DATA_BLOCK "HF4_Sum_SCtrl"	// DB 6040
VERSION : 0.1
  STRUCT
   SDPH_1_SCtrl : WORD ;
   SDPH_2_SCtrl : WORD ;
   SDPH_3_SCtrl : WORD ;
   SDPH_4_SCtrl : WORD ;
   SDPH_5_SCtrl : WORD ;
   SDPH_6_SCtrl : WORD ;
   SDPH_7_SCtrl : WORD ;
   SDPH_8_SCtrl : WORD ;
   SDPH_9_SCtrl : WORD ;
   SDPH_10_SCtrl : WORD ;
   SB_1_SCtrl : WORD ;
   SB_2_SCtrl : WORD ;
   SB_3_SCtrl : WORD ;
   SB_4_SCtrl : WORD ;
   SB_5_SCtrl : WORD ;
   SB_6_SCtrl : WORD ;
   SB_7_SCtrl : WORD ;
   SB_8_SCtrl : WORD ;
   SB_9_SCtrl : WORD ;
   SB_10_SCtrl : WORD ;
   SB_11_SCtrl : WORD ;
   SB_12_SCtrl : WORD ;
   SB_13_SCtrl : WORD ;
   SB_14_SCtrl : WORD ;
   SB_15_SCtrl : WORD ;
   SB_16_SCtrl : WORD ;
   SB_17_SCtrl : WORD ;
   SB_18_SCtrl : WORD ;
   KT_A1_SCtrl : WORD ;
   HPF_A1_SCtrl : WORD ;
   DTS_A1_SCtrl : WORD ;
   DTS_A2_SCtrl : WORD ;
   DTS_A3_SCtrl : WORD ;
   DTS_A4_SCtrl : WORD ;
   DTS_A5_SCtrl : WORD ;
   DTS_A6_SCtrl : WORD ;
   DTS_A7_SCtrl : WORD ;
   DTS_A8_SCtrl : WORD ;
   DTS_A9_SCtrl : WORD ;
   DTS_A10_SCtrl : WORD ;
   TVF_A1_SCtrl : WORD ;
   TVF_A2_SCtrl : WORD ;
   UOF_A1_SCtrl : WORD ;
   DM_A1_SCtrl : WORD ;
   DM_A2_SCtrl : WORD ;
   DM_A3_SCtrl : WORD ;
   DM_A4_SCtrl : WORD ;
   DM_A5_SCtrl : WORD ;
   DM_A6_SCtrl : WORD ;
   DM_A7_SCtrl : WORD ;
   DM_A8_SCtrl : WORD ;
   DM_A9_SCtrl : WORD ;
   DM_A10_SCtrl : WORD ;
   U0F_DT_A1_SCtrl : WORD ;
   U0F_DT_A2_SCtrl : WORD ;
   U0F_DT_A3_SCtrl : WORD ;
   U0F_DT_A4_SCtrl : WORD ;
   U0F_DT_A5_SCtrl : WORD ;
   U0F_DT_A6_SCtrl : WORD ;
   K1_XK_A1_SCtrl : WORD ;
   K1_HPF_A1_SCtrl : WORD ;
   K1_DTS_A1_SCtrl : WORD ;
   K1_DTS_A2_SCtrl : WORD ;
   K1_DTS_A3_SCtrl : WORD ;
   K2_XK_A1_SCtrl : WORD ;
   K2_HPF_A1_SCtrl : WORD ;
   K2_DTS_A1_SCtrl : WORD ;
   K2_DTS_A2_SCtrl : WORD ;
   K2_DTS_A3_SCtrl : WORD ;
   K3_XK_A1_SCtrl : WORD ;
   K3_HPF_A1_SCtrl : WORD ;
   K3_DTS_A1_SCtrl : WORD ;
   K3_DTS_A2_SCtrl : WORD ;
   K3_DTS_A3_SCtrl : WORD ;
   K4_XK_A1_SCtrl : WORD ;
   K4_HPF_A1_SCtrl : WORD ;
   K4_DTS_A1_SCtrl : WORD ;
   K4_DTS_A2_SCtrl : WORD ;
   K4_DTS_A3_SCtrl : WORD ;
   K5_XK_A1_SCtrl : WORD ;
   K5_HPF_A1_SCtrl : WORD ;
   K5_DTS_A1_SCtrl : WORD ;
   K5_DTS_A2_SCtrl : WORD ;
   K5_DTS_A3_SCtrl : WORD ;
   K6_XK_A1_SCtrl : WORD ;
   K6_HPF_A1_SCtrl : WORD ;
   K6_DTS_A1_SCtrl : WORD ;
   K6_DTS_A2_SCtrl : WORD ;
   K6_DTS_A3_SCtrl : WORD ;
   K7_XK_A1_SCtrl : WORD ;
   K7_HPF_A1_SCtrl : WORD ;
   K7_DTS_A1_SCtrl : WORD ;
   K7_DTS_A2_SCtrl : WORD ;
   K7_DTS_A3_SCtrl : WORD ;
   T1_XSF_A1_SCtrl : WORD ;
   T1_XPF_A1_SCtrl : WORD ;
   T1_D_A1_SCtrl : WORD ;
   T1_D_A2_SCtrl : WORD ;
   T2_XSF_A1_SCtrl : WORD ;
   T2_XPF_A1_SCtrl : WORD ;
   T2_D_A1_SCtrl : WORD ;
   T2_D_A2_SCtrl : WORD ;
   T3_XSF_A1_SCtrl : WORD ;
   T3_XPF_A1_SCtrl : WORD ;
   T3_D_A1_SCtrl : WORD ;
   T3_D_A2_SCtrl : WORD ;
   T4_XSF_A1_SCtrl : WORD ;
   T4_XPF_A1_SCtrl : WORD ;
   T4_D_A1_SCtrl : WORD ;
   T4_D_A2_SCtrl : WORD ;
   T5_XSF_A1_SCtrl : WORD ;
   T5_XPF_A1_SCtrl : WORD ;
   T5_D_A1_SCtrl : WORD ;
   T5_D_A2_SCtrl : WORD ;
   T6_XSF_A1_SCtrl : WORD ;
   T6_XPF_A1_SCtrl : WORD ;
   T6_D_A1_SCtrl : WORD ;
   T6_D_A2_SCtrl : WORD ;
   T7_XSF_A1_SCtrl : WORD ;
   T7_XPF_A1_SCtrl : WORD ;
   T7_D_A1_SCtrl : WORD ;
   T7_D_A2_SCtrl : WORD ;
   T8_XSF_A1_SCtrl : WORD ;
   T8_XPF_A1_SCtrl : WORD ;
   T8_XSF_A2_SCtrl : WORD ;
   T8_XPF_A2_SCtrl : WORD ;
   T8_D_A1_SCtrl : WORD ;
   T8_D_A2_SCtrl : WORD ;
   T8_D_A3_SCtrl : WORD ;
   T8_D_A4_SCtrl : WORD ;
   T8_D_A5_SCtrl : WORD ;
   T8_D_A6_SCtrl : WORD ;
   T8_D_A7_SCtrl : WORD ;
   T8_D_A8_SCtrl : WORD ;
   T8_D_A9_SCtrl : WORD ;
   T8_D_A10_SCtrl : WORD ;
   RF_A_SCtrl : WORD ;
   DT_RF_A1_SCtrl : WORD ;
   KT_B1_SCtrl : WORD ;
   HPF_B1_SCtrl : WORD ;
   DTS_B1_SCtrl : WORD ;
   DTS_B2_SCtrl : WORD ;
   DTS_B3_SCtrl : WORD ;
   DTS_B4_SCtrl : WORD ;
   DTS_B5_SCtrl : WORD ;
   DTS_B6_SCtrl : WORD ;
   DTS_B7_SCtrl : WORD ;
   DTS_B8_SCtrl : WORD ;
   DTS_B9_SCtrl : WORD ;
   DTS_B10_SCtrl : WORD ;
   TVF_B1_SCtrl : WORD ;
   TVF_B2_SCtrl : WORD ;
   UOF_B1_SCtrl : WORD ;
   DM_B1_SCtrl : WORD ;
   DM_B2_SCtrl : WORD ;
   DM_B3_SCtrl : WORD ;
   DM_B4_SCtrl : WORD ;
   DM_B5_SCtrl : WORD ;
   DM_B6_SCtrl : WORD ;
   DM_B7_SCtrl : WORD ;
   DM_B8_SCtrl : WORD ;
   DM_B9_SCtrl : WORD ;
   DM_B10_SCtrl : WORD ;
   U0F_DT_B1_SCtrl : WORD ;
   U0F_DT_B2_SCtrl : WORD ;
   U0F_DT_B3_SCtrl : WORD ;
   U0F_DT_B4_SCtrl : WORD ;
   U0F_DT_B5_SCtrl : WORD ;
   U0F_DT_B6_SCtrl : WORD ;
   K1_XK_B1_SCtrl : WORD ;
   K1_HPF_B1_SCtrl : WORD ;
   K1_DTS_B1_SCtrl : WORD ;
   K1_DTS_B2_SCtrl : WORD ;
   K1_DTS_B3_SCtrl : WORD ;
   K2_XK_B1_SCtrl : WORD ;
   K2_HPF_B1_SCtrl : WORD ;
   K2_DTS_B1_SCtrl : WORD ;
   K2_DTS_B2_SCtrl : WORD ;
   K2_DTS_B3_SCtrl : WORD ;
   K3_XK_B1_SCtrl : WORD ;
   K3_HPF_B1_SCtrl : WORD ;
   K3_DTS_B1_SCtrl : WORD ;
   K3_DTS_B2_SCtrl : WORD ;
   K3_DTS_B3_SCtrl : WORD ;
   K4_XK_B1_SCtrl : WORD ;
   K4_HPF_B1_SCtrl : WORD ;
   K4_DTS_B1_SCtrl : WORD ;
   K4_DTS_B2_SCtrl : WORD ;
   K4_DTS_B3_SCtrl : WORD ;
   K5_XK_B1_SCtrl : WORD ;
   K5_HPF_B1_SCtrl : WORD ;
   K5_DTS_B1_SCtrl : WORD ;
   K5_DTS_B2_SCtrl : WORD ;
   K5_DTS_B3_SCtrl : WORD ;
   K6_XK_B1_SCtrl : WORD ;
   K6_HPF_B1_SCtrl : WORD ;
   K6_DTS_B1_SCtrl : WORD ;
   K6_DTS_B2_SCtrl : WORD ;
   K6_DTS_B3_SCtrl : WORD ;
   K7_XK_B1_SCtrl : WORD ;
   K7_HPF_B1_SCtrl : WORD ;
   K7_DTS_B1_SCtrl : WORD ;
   K7_DTS_B2_SCtrl : WORD ;
   K7_DTS_B3_SCtrl : WORD ;
   T1_XSF_B1_SCtrl : WORD ;
   T1_XPF_B1_SCtrl : WORD ;
   T1_D_B1_SCtrl : WORD ;
   T1_D_B2_SCtrl : WORD ;
   T2_XSF_B1_SCtrl : WORD ;
   T2_XPF_B1_SCtrl : WORD ;
   T2_D_B1_SCtrl : WORD ;
   T2_D_B2_SCtrl : WORD ;
   T3_XSF_B1_SCtrl : WORD ;
   T3_XPF_B1_SCtrl : WORD ;
   T3_D_B1_SCtrl : WORD ;
   T3_D_B2_SCtrl : WORD ;
   T4_XSF_B1_SCtrl : WORD ;
   T4_XPF_B1_SCtrl : WORD ;
   T4_D_B1_SCtrl : WORD ;
   T4_D_B2_SCtrl : WORD ;
   T5_XSF_B1_SCtrl : WORD ;
   T5_XPF_B1_SCtrl : WORD ;
   T5_D_B1_SCtrl : WORD ;
   T5_D_B2_SCtrl : WORD ;
   T6_XSF_B1_SCtrl : WORD ;
   T6_XPF_B1_SCtrl : WORD ;
   T6_D_B1_SCtrl : WORD ;
   T6_D_B2_SCtrl : WORD ;
   T7_XSF_B1_SCtrl : WORD ;
   T7_XPF_B1_SCtrl : WORD ;
   T7_D_B1_SCtrl : WORD ;
   T7_D_B2_SCtrl : WORD ;
   T8_XSF_B1_SCtrl : WORD ;
   T8_XPF_B1_SCtrl : WORD ;
   T8_XSF_B2_SCtrl : WORD ;
   T8_XPF_B2_SCtrl : WORD ;
   T8_D_B1_SCtrl : WORD ;
   T8_D_B2_SCtrl : WORD ;
   T8_D_B3_SCtrl : WORD ;
   T8_D_B4_SCtrl : WORD ;
   T8_D_B5_SCtrl : WORD ;
   T8_D_B6_SCtrl : WORD ;
   T8_D_B7_SCtrl : WORD ;
   T8_D_B8_SCtrl : WORD ;
   T8_D_B9_SCtrl : WORD ;
   T8_D_B10_SCtrl : WORD ;
   RF_B_SCtrl : WORD ;
   DT_RF_B1_SCtrl : WORD ;
   YL_01_SCtrl : WORD ;
   YL_02_SCtrl : WORD ;
   YL_03_SCtrl : WORD ;
   YL_04_SCtrl : WORD ;
   EPSA_WLE_1_SCtrl : WORD ;
   EPSA_WLE_2_SCtrl : WORD ;
   EPSA_WLE_3_SCtrl : WORD ;
   EPSA_WLE_4_SCtrl : WORD ;
   EPSA_WLE_5_SCtrl : WORD ;
   EPSA_WLE_6_SCtrl : WORD ;
   EPSA_WLE_7_SCtrl : WORD ;
   EPSA_WLE_8_SCtrl : WORD ;
   EPSB_WLE_1_SCtrl : WORD ;
   EPSB_WLE_2_SCtrl : WORD ;
   EPSB_WLE_3_SCtrl : WORD ;
   EPSB_WLE_4_SCtrl : WORD ;
   EPSB_WLE_5_SCtrl : WORD ;
   EPSB_WLE_6_SCtrl : WORD ;
   EPSB_WLE_7_SCtrl : WORD ;
   EPSB_WLE_8_SCtrl : WORD ;
   XFDF_1_SCtrl : WORD ;
   XFDF_2_SCtrl : WORD ;
   XFDF_3_SCtrl : WORD ;
   XFDF_4_SCtrl : WORD ;
   VRV_SCtrl : WORD ;
   LSQK_SCtrl : WORD ;
   ZNZM_SCtrl : WORD ;
   adb_ZNZM_SENES_CTRL : WORD ;
   TIME_SET : WORD ;
   AP_WP1_SCtrl : WORD ;
   AP_WP2_SCtrl : WORD ;
   AP_WP3_SCtrl : WORD ;
   AP_WP4_SCtrl : WORD ;
   AP_WP5_SCtrl : WORD ;
   T1_XSF_A2_SCtrl : WORD ;
   T1_XPF_A2_SCtrl : WORD ;
   T1_D_A3_SCtrl : WORD ;
   T1_D_A4_SCtrl : WORD ;
   T1_D_A5_SCtrl : WORD ;
   T1_XSF_B2_SCtrl : WORD ;
   T1_XPF_B2_SCtrl : WORD ;
   T1_D_B3_SCtrl : WORD ;
   T1_D_B4_SCtrl : WORD ;
   T1_D_B5_SCtrl : WORD ;
   T9_XSF_A1_SCtrl : WORD ;
   T9_XPF_A1_SCtrl : WORD ;
   T9_XSF_A2_SCtrl : WORD ;
   T9_XPF_A2_SCtrl : WORD ;
   T9_D_A1_SCtrl : WORD ;
   T9_D_A2_SCtrl : WORD ;
   T9_D_A3_SCtrl : WORD ;
   T9_D_A4_SCtrl : WORD ;
   T9_D_A5_SCtrl : WORD ;
   T9_D_A6_SCtrl : WORD ;
   T9_D_A7_SCtrl : WORD ;
   T9_D_A8_SCtrl : WORD ;
   T9_D_A9_SCtrl : WORD ;
   T9_D_A10_SCtrl : WORD ;
   T9_XSF_B1_SCtrl : WORD ;
   T9_XPF_B1_SCtrl : WORD ;
   T9_XSF_B2_SCtrl : WORD ;
   T9_XPF_B2_SCtrl : WORD ;
   T9_D_B1_SCtrl : WORD ;
   T9_D_B2_SCtrl : WORD ;
   T9_D_B3_SCtrl : WORD ;
   T9_D_B4_SCtrl : WORD ;
   T9_D_B5_SCtrl : WORD ;
   T9_D_B6_SCtrl : WORD ;
   T9_D_B7_SCtrl : WORD ;
   T9_D_B8_SCtrl : WORD ;
   T9_D_B9_SCtrl : WORD ;
   T9_D_B10_SCtrl : WORD ;
   T10_XSF_A1_SCtrl : WORD ;
   T10_XPF_A1_SCtrl : WORD ;
   T10_XSF_A2_SCtrl : WORD ;
   T10_XPF_A2_SCtrl : WORD ;
   T10_D_A1_SCtrl : WORD ;
   T10_D_A2_SCtrl : WORD ;
   T10_D_A3_SCtrl : WORD ;
   T10_D_A4_SCtrl : WORD ;
   T10_D_A5_SCtrl : WORD ;
   T10_D_A6_SCtrl : WORD ;
   T10_D_A7_SCtrl : WORD ;
   T10_D_A8_SCtrl : WORD ;
   T10_D_A9_SCtrl : WORD ;
   T10_D_A10_SCtrl : WORD ;
   T10_XSF_B1_SCtrl : WORD ;
   T10_XPF_B1_SCtrl : WORD ;
   T10_XSF_B2_SCtrl : WORD ;
   T10_XPF_B2_SCtrl : WORD ;
   T10_D_B1_SCtrl : WORD ;
   T10_D_B2_SCtrl : WORD ;
   T10_D_B3_SCtrl : WORD ;
   T10_D_B4_SCtrl : WORD ;
   T10_D_B5_SCtrl : WORD ;
   T10_D_B6_SCtrl : WORD ;
   T10_D_B7_SCtrl : WORD ;
   T10_D_B8_SCtrl : WORD ;
   T10_D_B9_SCtrl : WORD ;
   T10_D_B10_SCtrl : WORD ;
   T11_XSF_A1_SCtrl : WORD ;
   T11_XPF_A1_SCtrl : WORD ;
   T11_XSF_A2_SCtrl : WORD ;
   T11_XPF_A2_SCtrl : WORD ;
   T11_D_A1_SCtrl : WORD ;
   T11_D_A2_SCtrl : WORD ;
   T11_D_A3_SCtrl : WORD ;
   T11_D_A4_SCtrl : WORD ;
   T11_D_A5_SCtrl : WORD ;
   T11_D_A6_SCtrl : WORD ;
   T11_D_A7_SCtrl : WORD ;
   T11_D_A8_SCtrl : WORD ;
   T11_D_A9_SCtrl : WORD ;
   T11_D_A10_SCtrl : WORD ;
   T11_XSF_B1_SCtrl : WORD ;
   T11_XPF_B1_SCtrl : WORD ;
   T11_XSF_B2_SCtrl : WORD ;
   T11_XPF_B2_SCtrl : WORD ;
   T11_D_B1_SCtrl : WORD ;
   T11_D_B2_SCtrl : WORD ;
   T11_D_B3_SCtrl : WORD ;
   T11_D_B4_SCtrl : WORD ;
   T11_D_B5_SCtrl : WORD ;
   T11_D_B6_SCtrl : WORD ;
   T11_D_B7_SCtrl : WORD ;
   T11_D_B8_SCtrl : WORD ;
   T11_D_B9_SCtrl : WORD ;
   T11_D_B10_SCtrl : WORD ;
   T12_XSF_A1_SCtrl : WORD ;
   T12_XPF_A1_SCtrl : WORD ;
   T12_XSF_A2_SCtrl : WORD ;
   T12_XPF_A2_SCtrl : WORD ;
   T12_D_A1_SCtrl : WORD ;
   T12_D_A2_SCtrl : WORD ;
   T12_D_A3_SCtrl : WORD ;
   T12_D_A4_SCtrl : WORD ;
   T12_D_A5_SCtrl : WORD ;
   T12_D_A6_SCtrl : WORD ;
   T12_D_A7_SCtrl : WORD ;
   T12_D_A8_SCtrl : WORD ;
   T12_D_A9_SCtrl : WORD ;
   T12_D_A10_SCtrl : WORD ;
   T12_XSF_B1_SCtrl : WORD ;
   T12_XPF_B1_SCtrl : WORD ;
   T12_XSF_B2_SCtrl : WORD ;
   T12_XPF_B2_SCtrl : WORD ;
   T12_D_B1_SCtrl : WORD ;
   T12_D_B2_SCtrl : WORD ;
   T12_D_B3_SCtrl : WORD ;
   T12_D_B4_SCtrl : WORD ;
   T12_D_B5_SCtrl : WORD ;
   T12_D_B6_SCtrl : WORD ;
   T12_D_B7_SCtrl : WORD ;
   T12_D_B8_SCtrl : WORD ;
   T12_D_B9_SCtrl : WORD ;
   T12_D_B10_SCtrl : WORD ;
   YL_05_SCTRL : ARRAY  [0 .. 272 ] OF WORD ;
   KT_A1_KpTm : INT ;
   KT_A1_KiTm : INT ;
   KT_A1_SPTm : INT ;
   KT_A1_OMS : INT ;
   HPF_A1_KpTm : INT ;
   HPF_A1_KiTm : INT ;
   HPF_A1_SPTm : INT ;
   HPF_A1_OMS : INT ;
   UOF_A1_KpTm : INT ;
   UOF_A1_KiTm : INT ;
   UOF_A1_SPTm : INT ;
   UOF_A1_OMS : INT ;
   KT_B1_KpTm : INT ;
   KT_B1_KiTm : INT ;
   KT_B1_SPTm : INT ;
   KT_B1_OMS : INT ;
   HPF_B1_KpTm : INT ;
   HPF_B1_KiTm : INT ;
   HPF_B1_SPTm : INT ;
   HPF_B1_OMS : INT ;
   UOF_B1_KpTm : INT ;
   UOF_B1_KiTm : INT ;
   UOF_B1_SPTm : INT ;
   UOF_B1_OMS : INT ;
   SDPH_1_KpTm : INT ;
   SDPH_1_KiTm : INT ;
   SDPH_1_SPTm : INT ;
   SDPH_1_OMS : INT ;
   SDPH_2_KpTm : INT ;
   SDPH_2_KiTm : INT ;
   SDPH_2_SPTm : INT ;
   SDPH_2_OMS : INT ;
   SDPH_3_KpTm : INT ;
   SDPH_3_KiTm : INT ;
   SDPH_3_SPTm : INT ;
   SDPH_3_OMS : INT ;
   SDPH_4_KpTm : INT ;
   SDPH_4_KiTm : INT ;
   SDPH_4_SPTm : INT ;
   SDPH_4_OMS : INT ;
   SDPH_5_KpTm : INT ;
   SDPH_5_KiTm : INT ;
   SDPH_5_SPTm : INT ;
   SDPH_5_OMS : INT ;
   SDPH_6_KpTm : INT ;
   SDPH_6_KiTm : INT ;
   SDPH_6_SPTm : INT ;
   SDPH_6_OMS : INT ;
   SDPH_7_KpTm : INT ;
   SDPH_7_KiTm : INT ;
   SDPH_7_SPTm : INT ;
   SDPH_7_OMS : INT ;
   SDPH_8_KpTm : INT ;
   SDPH_8_KiTm : INT ;
   SDPH_8_SPTm : INT ;
   SDPH_8_OMS : INT ;
   SDPH_9_KpTm : INT ;
   SDPH_9_KiTm : INT ;
   SDPH_9_SPTm : INT ;
   SDPH_9_OMS : INT ;
   SDPH_10_KpTm : INT ;
   SDPH_10_KiTm : INT ;
   SDPH_10_SPTm : INT ;
   SDPH_10_OMS : INT ;
   ZNZM_SENES_CTRL : INT ;	//新增
  END_STRUCT ;	
BEGIN
END_DATA_BLOCK

DATA_BLOCK DB 6868
VERSION : 0.0
"HF3_MODE_PRO"
BEGIN
END_DATA_BLOCK

DATA_BLOCK "HF4_Mode_DB"	// DB 7004
VERSION : 0.0
  STRUCT 	//A端大系统模式控制
   KT_A1_Mctrl : ARRAY  [0 .. 3 ] OF BOOL ;
   HPF_A1_Mctrl : ARRAY  [0 .. 3 ] OF BOOL ;
   DTS_A1_Mctrl : ARRAY  [0 .. 3 ] OF BOOL ;
   DTS_A2_Mctrl : ARRAY  [0 .. 3 ] OF BOOL ;
   DTS_A3_Mctrl : ARRAY  [0 .. 3 ] OF BOOL ;
   DTS_A4_Mctrl : ARRAY  [0 .. 3 ] OF BOOL ;
   DTS_A5_Mctrl : ARRAY  [0 .. 3 ] OF BOOL ;
   DTS_A6_Mctrl : ARRAY  [0 .. 3 ] OF BOOL ;	//SDPF_A2_Mctrl:ARRAY [0..3]OF BOOL;
//A端隧道通风系统模式控制
   TVF_A1_Mctrl : ARRAY  [0 .. 3 ] OF BOOL ;
   TVF_A2_Mctrl : ARRAY  [0 .. 3 ] OF BOOL ;
   UOF_A1_Mctrl : ARRAY  [0 .. 3 ] OF BOOL ;
   DM_A1_Mctrl : ARRAY  [0 .. 3 ] OF BOOL ;
   DM_A2_Mctrl : ARRAY  [0 .. 3 ] OF BOOL ;
   DM_A3_Mctrl : ARRAY  [0 .. 3 ] OF BOOL ;
   DM_A4_Mctrl : ARRAY  [0 .. 3 ] OF BOOL ;
   DM_A5_Mctrl : ARRAY  [0 .. 3 ] OF BOOL ;
   DM_A6_Mctrl : ARRAY  [0 .. 3 ] OF BOOL ;
   DM_A7_Mctrl : ARRAY  [0 .. 3 ] OF BOOL ;
   DM_A8_Mctrl : ARRAY  [0 .. 3 ] OF BOOL ;
   UOF_DT_A1_Mctrl : ARRAY  [0 .. 3 ] OF BOOL ;
   UOF_DT_A2_Mctrl : ARRAY  [0 .. 3 ] OF BOOL ;
   UOF_DT_A3_Mctrl : ARRAY  [0 .. 3 ] OF BOOL ;
   UOF_DT_A4_Mctrl : ARRAY  [0 .. 3 ] OF BOOL ;
   AT_ZSL1_Mctrl : ARRAY  [0 .. 3 ] OF BOOL ;
   AT_ZSL2_Mctrl : ARRAY  [0 .. 3 ] OF BOOL ;
   AT_ZSL3_Mctrl : ARRAY  [0 .. 3 ] OF BOOL ;
   AT_ZSL4_Mctrl : ARRAY  [0 .. 3 ] OF BOOL ;	//A1小系统模式控制
   K4_XK_A1_Mctrl : ARRAY  [0 .. 3 ] OF BOOL ;
   K4_HPF_A1_Mctrl : ARRAY  [0 .. 3 ] OF BOOL ;
   K4_DTS_A1_Mctrl : ARRAY  [0 .. 3 ] OF BOOL ;
   K4_DTS_A2_Mctrl : ARRAY  [0 .. 3 ] OF BOOL ;
   K4_DTS_A3_Mctrl : ARRAY  [0 .. 3 ] OF BOOL ;	//A2小系统模式控制
   T6_XSF_A1_Mctrl : ARRAY  [0 .. 3 ] OF BOOL ;
   T6_XPF_A1_Mctrl : ARRAY  [0 .. 3 ] OF BOOL ;
   T6_D_A1_Mctrl : ARRAY  [0 .. 3 ] OF BOOL ;
   T6_D_A2_Mctrl : ARRAY  [0 .. 3 ] OF BOOL ;	//A3小系统模式控制
   T7_XPF_A1_Mctrl : ARRAY  [0 .. 3 ] OF BOOL ;
   T7_D_A1_Mctrl : ARRAY  [0 .. 3 ] OF BOOL ;
  END_STRUCT ;	
BEGIN
END_DATA_BLOCK

DATA_BLOCK "Maste_To_Slave_Mod_DB"	// DB 7005
VERSION : 0.1
  STRUCT
   BigA_Mode : ARRAY  [0 .. 15 ] OF BOOL ;
   TubA_Mode : ARRAY  [0 .. 15 ] OF BOOL ;
   A1_Mode : ARRAY  [0 .. 15 ] OF BOOL ;
   A2_Mode : ARRAY  [0 .. 15 ] OF BOOL ;
   A3_Mode : ARRAY  [0 .. 15 ] OF BOOL ;
   A4_Mode : ARRAY  [0 .. 15 ] OF BOOL ;
   A5_Mode : ARRAY  [0 .. 15 ] OF BOOL ;
   A6_Mode : ARRAY  [0 .. 15 ] OF BOOL ;
   A7_Mode : ARRAY  [0 .. 15 ] OF BOOL ;
   A8_Mode : ARRAY  [0 .. 15 ] OF BOOL ;
   A9_Mode : ARRAY  [0 .. 15 ] OF BOOL ;
   A10_Mode : ARRAY  [0 .. 15 ] OF BOOL ;
   A11_Mode : ARRAY  [0 .. 15 ] OF BOOL ;
   A12_Mode : ARRAY  [0 .. 15 ] OF BOOL ;
   BigA_ModeRefuse : BOOL ;
   TubA_ModeRefuse : BOOL ;	//B12_ModeRefuse:bool;
   BigA_All : ARRAY  [0 .. 15 ] OF BOOL ;
   TubA_All : ARRAY  [0 .. 15 ] OF BOOL ;
   A1_All : ARRAY  [0 .. 15 ] OF BOOL ;
   A2_All : ARRAY  [0 .. 15 ] OF BOOL ;
   A3_All : ARRAY  [0 .. 15 ] OF BOOL ;
   A4_All : ARRAY  [0 .. 15 ] OF BOOL ;
   A5_All : ARRAY  [0 .. 15 ] OF BOOL ;
   A6_All : ARRAY  [0 .. 15 ] OF BOOL ;
   A7_All : ARRAY  [0 .. 15 ] OF BOOL ;
   A8_All : ARRAY  [0 .. 15 ] OF BOOL ;
   A9_All : ARRAY  [0 .. 15 ] OF BOOL ;
   A10_All : ARRAY  [0 .. 15 ] OF BOOL ;
   A11_All : ARRAY  [0 .. 15 ] OF BOOL ;
   A12_All : ARRAY  [0 .. 15 ] OF BOOL ;
   FireAlarm : BOOL ;	//火灾信号
   BlockAlarm : BOOL ;	//阻塞信号
   BigA_Act_Mode : STRUCT
    BigA_Mode_Num : INT ;
    WORD0 : WORD ;
    WORD1 : WORD ;
    WORD2 : WORD ;
    WORD3 : WORD ;
    WORD4 : WORD ;
    WORD5 : WORD ;
    WORD6 : WORD ;
    WORD7 : WORD ;
   END_STRUCT ;
   TubA_Act_Mode : STRUCT
    TubA_Mode_Num : INT ;
    WORD0 : WORD ;
    WORD1 : WORD ;
    WORD2 : WORD ;
    WORD3 : WORD ;
    WORD4 : WORD ;
    WORD5 : WORD ;
    WORD6 : WORD ;
    WORD7 : WORD ;
   END_STRUCT ;
   A1_Act_Mode : STRUCT
    A1_Mode_Num : INT ;
    WORD0 : WORD ;
    WORD1 : WORD ;
    WORD2 : WORD ;
    WORD3 : WORD ;
    WORD4 : WORD ;
    WORD5 : WORD ;
    WORD6 : WORD ;
    WORD7 : WORD ;
   END_STRUCT ;
   A2_Act_Mode : STRUCT
    A2_Mode_Num : INT ;
    WORD0 : WORD ;
    WORD1 : WORD ;
    WORD2 : WORD ;
    WORD3 : WORD ;
    WORD4 : WORD ;
    WORD5 : WORD ;
    WORD6 : WORD ;
    WORD7 : WORD ;
   END_STRUCT ;
   A3_Act_Mode : STRUCT
    A3_Mode_Num : INT ;
    WORD0 : WORD ;
    WORD1 : WORD ;
    WORD2 : WORD ;
    WORD3 : WORD ;
    WORD4 : WORD ;
    WORD5 : WORD ;
    WORD6 : WORD ;
    WORD7 : WORD ;
   END_STRUCT ;
   A4_Act_Mode : STRUCT
    A4_Mode_Num : INT ;
    WORD0 : WORD ;
    WORD1 : WORD ;
    WORD2 : WORD ;
    WORD3 : WORD ;
    WORD4 : WORD ;
    WORD5 : WORD ;
    WORD6 : WORD ;
    WORD7 : WORD ;
   END_STRUCT ;
   A5_Act_Mode : STRUCT
    A5_Mode_Num : INT ;
    WORD0 : WORD ;
    WORD1 : WORD ;
    WORD2 : WORD ;
    WORD3 : WORD ;
    WORD4 : WORD ;
    WORD5 : WORD ;
    WORD6 : WORD ;
    WORD7 : WORD ;
   END_STRUCT ;
   A6_Act_Mode : STRUCT
    A6_Mode_Num : INT ;
    WORD0 : WORD ;
    WORD1 : WORD ;
    WORD2 : WORD ;
    WORD3 : WORD ;
    WORD4 : WORD ;
    WORD5 : WORD ;
    WORD6 : WORD ;
    WORD7 : WORD ;
   END_STRUCT ;
   A7_Act_Mode : STRUCT
    A7_Mode_Num : INT ;
    WORD0 : WORD ;
    WORD1 : WORD ;
    WORD2 : WORD ;
    WORD3 : WORD ;
    WORD4 : WORD ;
    WORD5 : WORD ;
    WORD6 : WORD ;
    WORD7 : WORD ;
   END_STRUCT ;
   A8_Act_Mode : STRUCT
    A8_Mode_Num : INT ;
    WORD0 : WORD ;
    WORD1 : WORD ;
    WORD2 : WORD ;
    WORD3 : WORD ;
    WORD4 : WORD ;
    WORD5 : WORD ;
    WORD6 : WORD ;
    WORD7 : WORD ;
   END_STRUCT ;
   A9_Act_Mode : STRUCT
    A9_Mode_Num : INT ;
    WORD0 : WORD ;
    WORD1 : WORD ;
    WORD2 : WORD ;
    WORD3 : WORD ;
    WORD4 : WORD ;
    WORD5 : WORD ;
    WORD6 : WORD ;
    WORD7 : WORD ;
   END_STRUCT ;
   A10_Act_Mode : STRUCT
    A10_Mode_Num : INT ;
    WORD0 : WORD ;
    WORD1 : WORD ;
    WORD2 : WORD ;
    WORD3 : WORD ;
    WORD4 : WORD ;
    WORD5 : WORD ;
    WORD6 : WORD ;
    WORD7 : WORD ;
   END_STRUCT ;
   A11_Act_Mode : STRUCT
    A11_Mode_Num : INT ;
    WORD0 : WORD ;
    WORD1 : WORD ;
    WORD2 : WORD ;
    WORD3 : WORD ;
    WORD4 : WORD ;
    WORD5 : WORD ;
    WORD6 : WORD ;
    WORD7 : WORD ;
   END_STRUCT ;
   A12_Act_Mode : STRUCT
    A12_Mode_Num : INT ;
    WORD0 : WORD ;
    WORD1 : WORD ;
    WORD2 : WORD ;
    WORD3 : WORD ;
    WORD4 : WORD ;
    WORD5 : WORD ;
    WORD6 : WORD ;
    WORD7 : WORD ;
   END_STRUCT ;
   H_P_ALL_Ctrl : WORD ;
  END_STRUCT ;	
BEGIN
END_DATA_BLOCK

DATA_BLOCK "MODE_REFUSE"	// DB 7006
VERSION : 0.0
  STRUCT
   BigA_ModeRefuse : BOOL ;	//大系统模式不符
   TubA_ModeRefuse : BOOL ;	//隧道通风模式不符
   A1_ModeRefuse : BOOL ;	//A1小系统模式不符
   A2_ModeRefuse : BOOL ;	//A2小系统模式不符
   A3_ModeRefuse : BOOL ;	//A3小系统模式不符
   A4_ModeRefuse : BOOL ;	//A4小系统模式不符
   A5_ModeRefuse : BOOL ;	//A5小系统模式不符
   A6_ModeRefuse : BOOL ;	//A6小系统模式不符
   A7_ModeRefuse : BOOL ;	//A7小系统模式不符
   A8_ModeRefuse : BOOL ;	//A8小系统模式不符
   A9_ModeRefuse : BOOL ;	//A9小系统模式不符
   A10_ModeRefuse : BOOL ;	//A10小系统模式不符
   A11_ModeRefuse : BOOL ;	//A11小系统模式不符
   A12_ModeRefuse : BOOL ;	//A12小系统模式不符
//A端大系统模式不符
   KT_A1_Refuse : BOOL ;
   HPF_A1_Refuse : BOOL ;
   DTS_A1_Refuse : BOOL ;
   DTS_A2_Refuse : BOOL ;
   DTS_A3_Refuse : BOOL ;
   DTS_A4_Refuse : BOOL ;
   DTS_A5_Refuse : BOOL ;
   DTS_A6_Refuse : BOOL ;
   DPH_A1_Refuse : BOOL ;	//A端隧道通风模式不符
   TVF_A1_Refuse : BOOL ;
   TVF_A2_Refuse : BOOL ;
   UOF_A1_Refuse : BOOL ;
   DM_A1_Refuse : BOOL ;
   DM_A2_Refuse : BOOL ;
   DM_A3_Refuse : BOOL ;
   DM_A4_Refuse : BOOL ;
   DM_A5_Refuse : BOOL ;
   DM_A6_Refuse : BOOL ;
   DM_A7_Refuse : BOOL ;
   DM_A8_Refuse : BOOL ;
   UOF_DT_A1_Refuse : BOOL ;
   UOF_DT_A2_Refuse : BOOL ;
   UOF_DT_A3_Refuse : BOOL ;
   UOF_DT_A4_Refuse : BOOL ;	//A1小系统
   K4_XK_A1_Refuse : BOOL ;
   K4_HPF_A1_Refuse : BOOL ;
   K4_DTS_A1_Refuse : BOOL ;
   K4_DTS_A2_Refuse : BOOL ;
   K4_DTS_A3_Refuse : BOOL ;	//A2小系统
   T6_XSF_A1_Refuse : BOOL ;
   T6_XPF_A1_Refuse : BOOL ;
   T6_D_A1_Refuse : BOOL ;
   T6_D_A2_Refuse : BOOL ;	//A3小系统
   T7_XPF_A1_Refuse : BOOL ;
   T7_D_A1_Refuse : BOOL ;
  END_STRUCT ;	
BEGIN
END_DATA_BLOCK

ORGANIZATION_BLOCK "HF3_Main_OB1"	// OB 1
TITLE = "B端主程序"
//程序主循环，调用所有子FC、FB程序段
VERSION : 0.1
VAR_TEMP
  OB1_EV_CLASS : BYTE ;	//Bits 0-3 = 1 (Coming event), Bits 4-7 = 1 (Event class 1)
  OB1_SCAN_1 : BYTE ;	//1 (Cold restart scan 1 of OB 1), 3 (Scan 2-n of OB 1)
  OB1_PRIORITY : BYTE ;	//Priority of OB Execution
  OB1_OB_NUMBR : BYTE ;	//1 (Organization block 1, OB1)
  OB1_RESERVED_1 : BYTE ;	//Reserved for system
  OB1_RESERVED_2 : BYTE ;	//Reserved for system
  OB1_PREV_CYCLE : INT ;	//Cycle time of previous OB1 scan (milliseconds)
  OB1_MIN_CYCLE : INT ;	//Minimum cycle time of OB1 (milliseconds)
  OB1_MAX_CYCLE : INT ;	//Maximum cycle time of OB1 (milliseconds)
  OB1_DATE_TIME : DATE_AND_TIME ;	//Date and time OB1 started
END_VAR
BEGIN
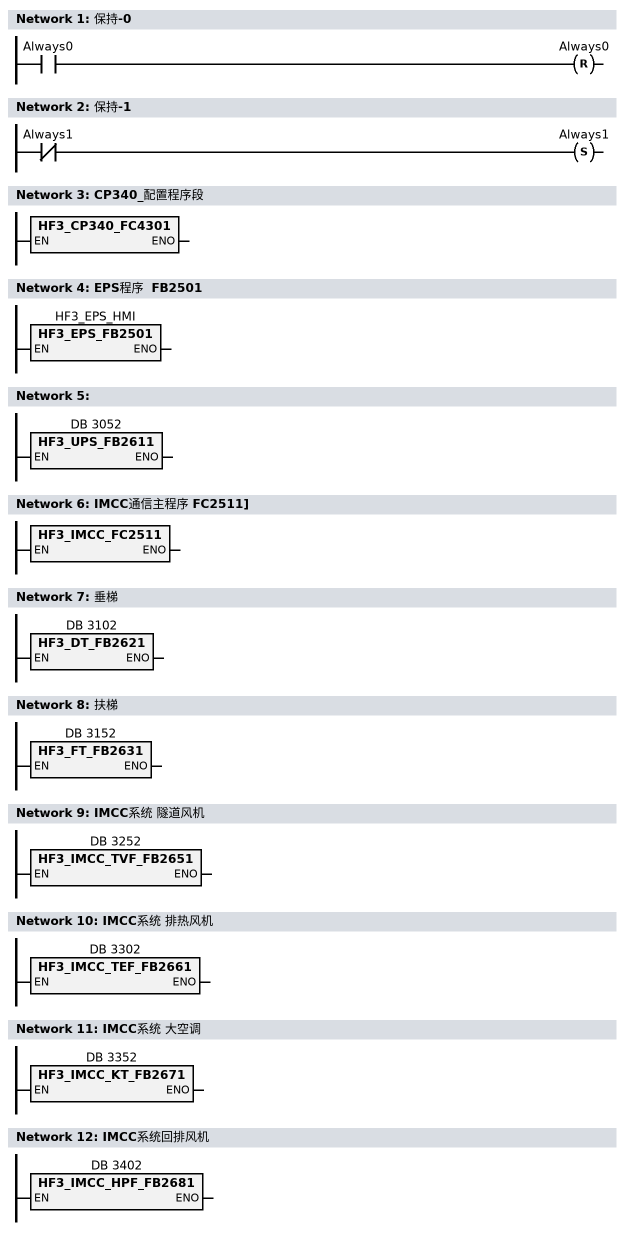
NETWORK
TITLE = 保持-0
      A     "Always0";
      R     "Always0";
NETWORK
TITLE = 保持-1
      AN    "Always1";
      S     "Always1";
NETWORK
TITLE = CP340_配置程序段
      CALL  "HF3_CP340_FC4301";
      NOP   0;
NETWORK
TITLE = EPS程序  FB2501
      CALL  "HF3_EPS_FB2501" , "HF3_EPS_HMI";
      NOP   0;
NETWORK
TITLE =
      CALL  "HF3_UPS_FB2611" , DB 3052;
      NOP   0;
NETWORK
TITLE = IMCC通信主程序 FC2511]
      CALL  "HF3_IMCC_FC2511";
      NOP   0;
NETWORK
TITLE = 垂梯
      CALL  "HF3_DT_FB2621" , DB 3102;
      NOP   0;
NETWORK
TITLE = 扶梯
      CALL  "HF3_FT_FB2631" , DB 3152;
      NOP   0;
NETWORK
TITLE = IMCC系统 隧道风机
      CALL  "HF3_IMCC_TVF_FB2651" , DB 3252;
      NOP   0;
NETWORK
TITLE = IMCC系统 排热风机
      CALL  "HF3_IMCC_TEF_FB2661" , DB 3302;
      NOP   0;
NETWORK
TITLE = IMCC系统 大空调
      CALL  "HF3_IMCC_KT_FB2671" , DB 3352;
      NOP   0;
NETWORK
TITLE = IMCC系统回排风机
      CALL  "HF3_IMCC_HPF_FB2681" , DB 3402;
      NOP   0;
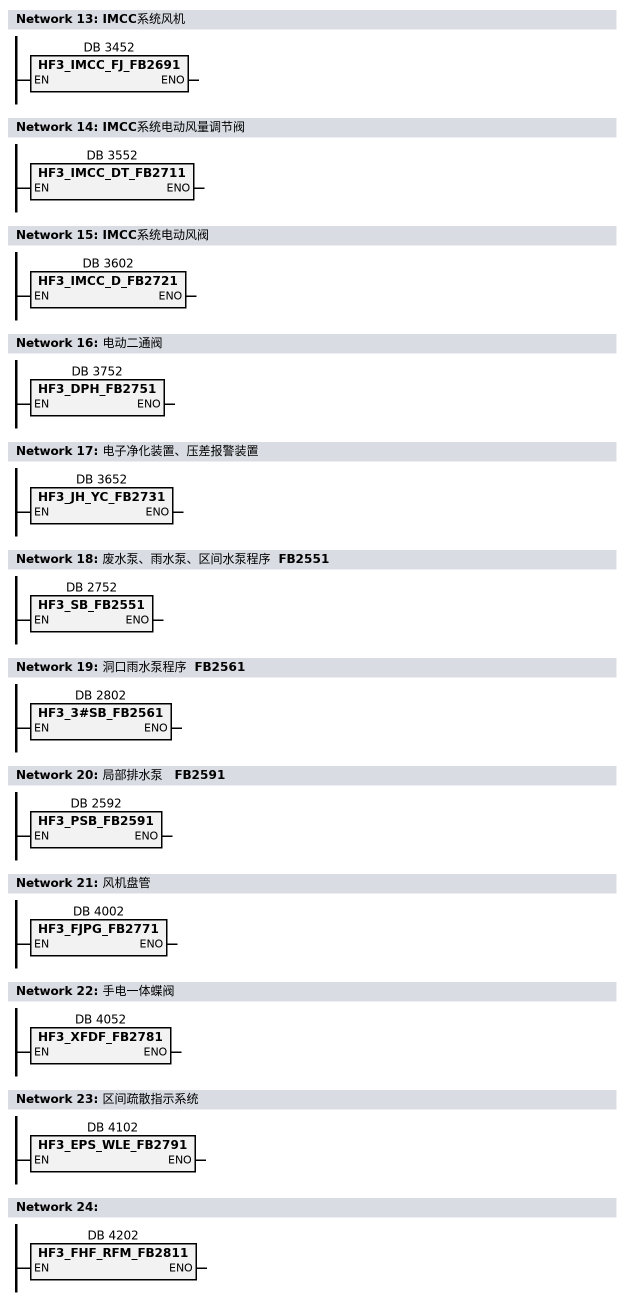
NETWORK
TITLE = IMCC系统风机
      CALL  "HF3_IMCC_FJ_FB2691" , DB 3452;
      NOP   0;
NETWORK
TITLE = IMCC系统电动风量调节阀
      CALL  "HF3_IMCC_DT_FB2711" , DB 3552;
      NOP   0;
NETWORK
TITLE = IMCC系统电动风阀
      CALL  "HF3_IMCC_D_FB2721" , DB 3602;
      NOP   0;
NETWORK
TITLE = 电动二通阀
      CALL  "HF3_DPH_FB2751" , DB 3752;
      NOP   0;
NETWORK
TITLE = 电子净化装置、压差报警装置
      CALL  "HF3_JH_YC_FB2731" , DB 3652;
      NOP   0;
NETWORK
TITLE = 废水泵、雨水泵、区间水泵程序  FB2551
      CALL  "HF3_SB_FB2551" , DB 2752;
      NOP   0;
NETWORK
TITLE = 洞口雨水泵程序  FB2561
      CALL  "HF3_3#SB_FB2561" , DB 2802;
      NOP   0;
NETWORK
TITLE = 局部排水泵　FB2591
      CALL  "HF3_PSB_FB2591" , DB 2592;
      NOP   0;
NETWORK
TITLE = 风机盘管
      CALL  "HF3_FJPG_FB2771" , DB 4002;
      NOP   0;
NETWORK
TITLE = 手电一体蝶阀
      CALL  "HF3_XFDF_FB2781" , DB 4052;
      NOP   0;
NETWORK
TITLE = 区间疏散指示系统
      CALL  "HF3_EPS_WLE_FB2791" , DB 4102;
      NOP   0;
NETWORK
TITLE =
      CALL  "HF3_FHF_RFM_FB2811" , DB 4202;
      NOP   0;
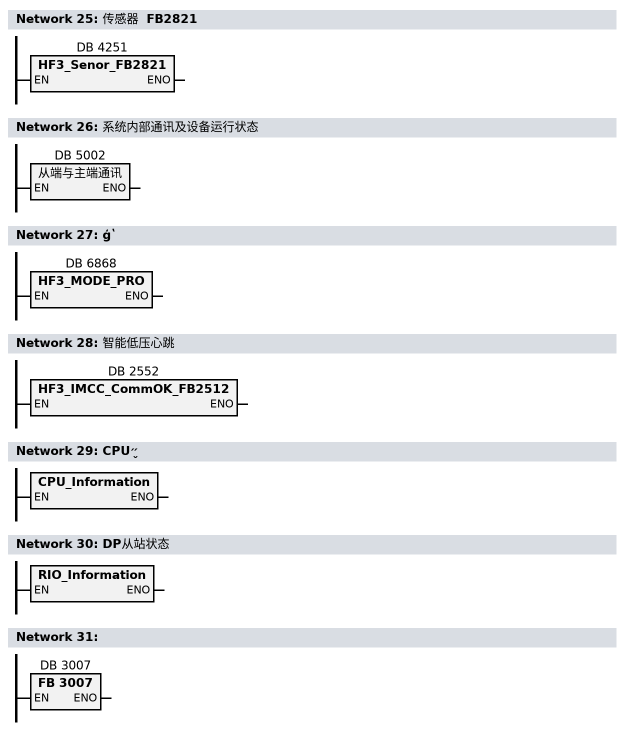
NETWORK
TITLE = 传感器  FB2821
      CALL  "HF3_Senor_FB2821" , DB 4251;
      NOP   0;
NETWORK
TITLE = 系统内部通讯及设备运行状态
      CALL  "从端与主端通讯" , DB 5002;
      NOP   0;
NETWORK
TITLE = ģʽ
      CALL  "HF3_MODE_PRO" , DB 6868;
      NOP   0;
NETWORK
TITLE = 智能低压心跳
      CALL  "HF3_IMCC_CommOK_FB2512" , DB 2552;
      NOP   0;
NETWORK
TITLE = CPU״̬
      CALL  "CPU_Information";
      NOP   0;
NETWORK
TITLE = DP从站状态
      CALL  "RIO_Information";
      NOP   0;
NETWORK
TITLE =
      CALL  FB 3007 , DB 3007;
      NOP   0;
END_ORGANIZATION_BLOCK

ORGANIZATION_BLOCK "CYC_INT5"	// OB 35
TITLE = "Cyclic Interrupt"
VERSION : 0.1
VAR_TEMP
  OB35_EV_CLASS : BYTE ;	//Bits 0-3 = 1 (Coming event), Bits 4-7 = 1 (Event class 1)
  OB35_STRT_INF : BYTE ;	//16#36 (OB 35 has started)
  OB35_PRIORITY : BYTE ;	//Priority of OB Execution
  OB35_OB_NUMBR : BYTE ;	//35 (Organization block 35, OB35)
  OB35_RESERVED_1 : BYTE ;	//Reserved for system
  OB35_RESERVED_2 : BYTE ;	//Reserved for system
  OB35_PHASE_OFFSET : WORD ;	//Phase offset (msec)
  OB35_RESERVED_3 : INT ;	//Reserved for system
  OB35_EXC_FREQ : INT ;	//Frequency of execution (msec)
  OB35_DATE_TIME : DATE_AND_TIME ;	//Date and time OB35 started
END_VAR
BEGIN
// (block stored without names or comments; labels and parameter names are numbered)
END_ORGANIZATION_BLOCK

ORGANIZATION_BLOCK "RED_I/O_FLT1"	// OB 70
TITLE = "Redundancy I/O Fault 1"
VERSION : 0.1
VAR_TEMP
  OB70_EV_CLASS : BYTE ;	//Event class 7, module inserted/removed (8/9)
  OB70_FLT_ID : BYTE ;	//Fault identifcation code
  OB70_PRIORITY : BYTE ;	//Priority of OB Execution
  OB70_OB_NUMBR : BYTE ;	//70 (Organization block 70, OB70)
  OB70_RESERVED_1 : WORD ;	//Reserved for system
  OB70_INFO_1 : WORD ;	//Info 1
  OB70_INFO_2 : WORD ;	//Info 2
  OB70_INFO_3 : WORD ;	//Info 3
  OB70_DATE_TIME : DATE_AND_TIME ;	//Date and time OB70 started
END_VAR
BEGIN
// (block stored without names or comments; labels and parameter names are numbered)
END_ORGANIZATION_BLOCK

ORGANIZATION_BLOCK "RED_FLT"	// OB 72
TITLE = "Redundancy Fault"
VERSION : 0.1
VAR_TEMP
  OB72_EV_CLASS : BYTE ;	//Event class 7, module inserted/removed (8/9)
  OB72_FLT_ID : BYTE ;	//Fault identifcation code
  OB72_PRIORITY : BYTE ;	//Priority of OB Execution
  OB72_OB_NUMBR : BYTE ;	//72 (Organization block 72, OB72)
  OB72_RESERVED_1 : WORD ;	//Reserved for system
  OB72_INFO_1 : WORD ;	//Info 1
  OB72_INFO_2 : WORD ;	//Info 2
  OB72_INFO_3 : WORD ;	//Info 3
  OB72_DATE_TIME : DATE_AND_TIME ;	//Date and time OB72 started
END_VAR
BEGIN
// (block stored without names or comments; labels and parameter names are numbered)
END_ORGANIZATION_BLOCK

ORGANIZATION_BLOCK "PS_FLT"	// OB 81
TITLE = "Power Supply Fault"
VERSION : 0.0
VAR_TEMP
  OB81_EV_CLASS : BYTE ;	//16#39, Event class 3, Entering event state, Internal fault event
  OB81_FLT_ID : BYTE ;	//16#XX, Fault identifcation code
  OB81_PRIORITY : BYTE ;	//Priority of OB Execution
  OB81_OB_NUMBR : BYTE ;	//81 (Organization block 81, OB81)
  OB81_RESERVED_1 : BYTE ;	//Reserved for system
  OB81_RESERVED_2 : BYTE ;	//Reserved for system
  OB81_RACK_CPU : WORD ;	//see online help (F1)
  OB81_RESERVED_3 : BYTE ;	//Reserved for system
  OB81_RESERVED_4 : BYTE ;	//Reserved for system
  OB81_RESERVED_5 : BYTE ;	//Reserved for system
  OB81_RESERVED_6 : BYTE ;	//Reserved for system
  OB81_DATE_TIME : DATE_AND_TIME ;	//Date and time OB81 started
END_VAR
BEGIN
NETWORK
TITLE =
      L     #OB81_FLT_ID;
      L     B#16#25;
      ==I;
      =     M 81.1;
      L     #OB81_EV_CLASS;
      L     B#16#39;
      ==I;
      =     M 81.2;
      A     M 81.1;
      A     M 81.2;
      S     M 81.0;
NETWORK
TITLE =
      L     #OB81_RACK_CPU;
      T     MW 90;
NETWORK
TITLE = Temporary placeholder variable
      AN    M 90.0;
      A     M 81.0;
      S     "HF3_PLC_Statu_ToHMI".R0_PS_ERROR;
      A     M 90.0;
      S     M 81.0;
      S     "HF3_PLC_Statu_ToHMI".R1_PS_ERROR;
NETWORK
TITLE =
      L     #OB81_EV_CLASS;
      L     B#16#38;
      ==I;
      =     M 81.6;
      A     M 81.6;
      R     M 81.0;
NETWORK
TITLE = Temporary placeholder variable
      AN    M 90.0;
      A     M 81.6;
      R     "HF3_PLC_Statu_ToHMI".R0_PS_ERROR;
      A     M 90.0;
      A     M 81.6;
      R     "HF3_PLC_Statu_ToHMI".R1_PS_ERROR;
END_ORGANIZATION_BLOCK

ORGANIZATION_BLOCK "I/O_FLT1"	// OB 82
TITLE = "Redundancy I/O Fault 1"
VERSION : 0.1
VAR_TEMP
  OB70_EV_CLASS : BYTE ;	//Event class 7, module inserted/removed (8/9)
  OB70_FLT_ID : BYTE ;	//Fault identifcation code
  OB70_PRIORITY : BYTE ;	//Priority of OB Execution
  OB70_OB_NUMBR : BYTE ;	//70 (Organization block 70, OB70)
  OB70_RESERVED_1 : WORD ;	//Reserved for system
  OB70_INFO_1 : WORD ;	//Info 1
  OB70_INFO_2 : WORD ;	//Info 2
  OB70_INFO_3 : WORD ;	//Info 3
  OB70_DATE_TIME : DATE_AND_TIME ;	//Date and time OB70 started
END_VAR
BEGIN
NETWORK
TITLE =
//DP_MASTERSYSTEM=1
      CALL  "DETAIL_DP_DIAG" , "DETAIL_DIAG_DB_RACK0" (
           DP_MASTERSYSTEM          := 1,
           EXTERNAL_DP_INTERFACE    := FALSE,
           MANUAL_MODE              := "DP_VAT".MANUAL_MODE,
           SINGLE_STEP_SLAVE        := "DP_VAT".SINGLE_STEP_SLAVE,
           SINGLE_STEP_ERROR        := "DP_VAT".SINGLE_STEP_ERROR,
           RESET                    := "DP_VAT".RESET,
           SINGLE_DIAG              := "DP_VAT".SINGLE_SLAVE_DIAG,
           SINGLE_DIAG_ADR          := "DP_VAT".SINGLE_DIAG_ADR,
           ALL_DP_SLAVES_OK         := "DP_VAT".ALL_SLAVES_OK,
           SUM_SLAVES_DIAG          := "DP_VAT".SUM_SLAVES_DIAG,
           SLAVE_ADR                := "DP_VAT".SLAVE_ADR,
           SLAVE_STATE              := "DP_VAT".SLAVE_STATE,
           SLAVE_IDENT_NO           := "DP_VAT".SLAVE_IDENT_NO,
           ERROR_NO                 := "DP_VAT".ERROR_NO,
           ERROR_TYPE               := "DP_VAT".ERROR_TYPE,
           MODULE_NO                := "DP_VAT".MODULE_NO,
           MODULE_STATE             := "DP_VAT".MODULE_STATE,
           CHANNEL_NO               := "DP_VAT".CHANNEL_NO,
           CHANNEL_TYPE             := "DP_VAT".CHANNEL_TYPE,
           CHANNEL_ERROR_CODE       := "DP_VAT".CHANNEL_ERROR_CODE,
           CHANNEL_ERROR_INFO_1     := "DP_VAT".CHANNEL_ERROR_INFO_1,
           CHANNEL_ERROR_INFO_2     := "DP_VAT".CHANNEL_ERROR_INFO_2,
           DIAG_COUNTER             := "DP_VAT".DIAG_COUNTER,
           DIAG_OVERFLOW            := "DP_VAT".DIAG_OVERFLOW,
           BUSY                     := "DP_VAT".BUSY);
      NOP   0;
NETWORK
TITLE =
//DP_MASTERSYSTEM=2
      CALL  "DETAIL_DP_DIAG" , "DETAIL_DIAG_DB_RACK1" (
           DP_MASTERSYSTEM          := 2,
           EXTERNAL_DP_INTERFACE    := FALSE,
           MANUAL_MODE              := "DP_VAT".MANUAL_MODE1,
           SINGLE_STEP_SLAVE        := "DP_VAT".SINGLE_STEP_SLAVE1,
           SINGLE_STEP_ERROR        := "DP_VAT".SINGLE_STEP_ERROR1,
           RESET                    := "DP_VAT".RESET1,
           SINGLE_DIAG              := "DP_VAT".SINGLE_SLAVE_DIAG1,
           SINGLE_DIAG_ADR          := "DP_VAT".SINGLE_DIAG_ADR1,
           ALL_DP_SLAVES_OK         := "DP_VAT".ALL_SLAVES_OK1,
           SUM_SLAVES_DIAG          := "DP_VAT".SUM_SLAVES_DIAG1,
           SLAVE_ADR                := "DP_VAT".SLAVE_ADR1,
           SLAVE_STATE              := "DP_VAT".SLAVE_STATE1,
           SLAVE_IDENT_NO           := "DP_VAT".SLAVE_IDENT_NO1,
           ERROR_NO                 := "DP_VAT".ERROR_NO1,
           ERROR_TYPE               := "DP_VAT".ERROR_TYPE1,
           MODULE_NO                := "DP_VAT".MODULE_NO1,
           MODULE_STATE             := "DP_VAT".MODULE_STATE1,
           CHANNEL_NO               := "DP_VAT".CHANNEL_NO1,
           CHANNEL_TYPE             := "DP_VAT".CHANNEL_TYPE1,
           CHANNEL_ERROR_CODE       := "DP_VAT".CHANNEL_ERROR_CODE1,
           CHANNEL_ERROR_INFO_1     := "DP_VAT".CHANNEL_ERROR_INFO_11,
           CHANNEL_ERROR_INFO_2     := "DP_VAT".CHANNEL_ERROR_INFO_21,
           DIAG_COUNTER             := "DP_VAT".DIAG_COUNTER1,
           DIAG_OVERFLOW            := "DP_VAT".DIAG_OVERFLOW1,
           BUSY                     := "DP_VAT".BUSY1);
      NOP   0;
END_ORGANIZATION_BLOCK

ORGANIZATION_BLOCK "I/O_FLT2"	// OB 83
TITLE = "I/O Point Fault"
VERSION : 0.1
VAR_TEMP
  OB83_EV_CLASS : BYTE ;	//16#38/39, Event class 3, module inserted/removed (8/9)
  OB83_FLT_ID : BYTE ;	//16#XX, Fault identifcation code
  OB83_PRIORITY : BYTE ;	//Priority of OB Execution
  OB83_OB_NUMBR : BYTE ;	//83 (Organization block 83, OB83)
  OB83_RESERVED_1 : BYTE ;	//Reserved for system
  OB83_MDL_ID : BYTE ;	//Input module (01010100), Output module (01010101)
  OB83_MDL_ADDR : WORD ;	//Base address of module with point fault
  OB83_RACK_NUM : INT ;	//Number of rack that has module with point fault
  OB83_MDL_TYPE : WORD ;	//Module type with point fault
  OB83_DATE_TIME : DATE_AND_TIME ;	//Date and time OB83 started
END_VAR
BEGIN
// (block stored without names or comments; labels and parameter names are numbered)
END_ORGANIZATION_BLOCK

ORGANIZATION_BLOCK "CPU_FLT"	// OB 84
TITLE = "CPU Fault"
VERSION : 0.1
VAR_TEMP
  OB84_EV_CLASS : BYTE ;	//16#38/39, Event class 3, module inserted/removed (8/9)
  OB84_FLT_ID : BYTE ;	//16#81, Fault identifcation code
  OB84_PRIORITY : BYTE ;	//Priority of OB Execution
  OB84_OB_NUMBR : BYTE ;	//84 (Organization block 84, OB84)
  OB84_RESERVED_1 : BYTE ;	//Reserved for system
  OB84_RESERVED_2 : BYTE ;	//Reserved for system
  OB84_RESERVED_3 : WORD ;	//Reserved for system
  OB84_RESERVED_4 : DWORD ;	//Reserved for system
  OB84_DATE_TIME : DATE_AND_TIME ;	//Date and time OB84 started
END_VAR
BEGIN
// (block stored without names or comments; labels and parameter names are numbered)
END_ORGANIZATION_BLOCK

ORGANIZATION_BLOCK "OBNL_FLT"	// OB 85
TITLE = "Organization Block (OB) Not Loaded Fault"
VERSION : 0.1
VAR_TEMP
  OB85_EV_CLASS : BYTE ;	//16#35 Event class 3
  OB85_FLT_ID : BYTE ;	//16#XX, Fault identification code
  OB85_PRIORITY : BYTE ;	//Priority of OB Execution
  OB85_OB_NUMBR : BYTE ;	//85 (Organization block 85, OB85)
  OB85_RESERVED_1 : BYTE ;	//Reserved for system
  OB85_RESERVED_2 : BYTE ;	//Reserved for system
  OB85_RESERVED_3 : INT ;	//Reserved for system
  OB85_ERR_EV_CLASS : BYTE ;	//Class of event causing error
  OB85_ERR_EV_NUM : BYTE ;	//Number of event causing error
  OB85_OB_PRIOR : BYTE ;	//Priority of OB causing error
  OB85_OB_NUM : BYTE ;	//Number of OB causing error
  OB85_DATE_TIME : DATE_AND_TIME ;	//Date and time OB85 started
END_VAR
BEGIN
// (block stored without names or comments; labels and parameter names are numbered)
END_ORGANIZATION_BLOCK

ORGANIZATION_BLOCK "RACK_FLT"	// OB 86
TITLE = "Redundancy I/O Fault 1"
VERSION : 0.1
VAR_TEMP
  OB70_EV_CLASS : BYTE ;	//Event class 7, module inserted/removed (8/9)
  OB70_FLT_ID : BYTE ;	//Fault identifcation code
  OB70_PRIORITY : BYTE ;	//Priority of OB Execution
  OB70_OB_NUMBR : BYTE ;	//70 (Organization block 70, OB70)
  OB70_RESERVED_1 : WORD ;	//Reserved for system
  OB70_INFO_1 : WORD ;	//Info 1
  OB70_INFO_2 : WORD ;	//Info 2
  OB70_INFO_3 : WORD ;	//Info 3
  OB70_DATE_TIME : DATE_AND_TIME ;	//Date and time OB70 started
END_VAR
BEGIN
NETWORK
TITLE =
//DP_MASTERSYSTEM=1
      CALL  "DETAIL_DP_DIAG" , "DETAIL_DIAG_DB_RACK0" (
           DP_MASTERSYSTEM          := 1,
           EXTERNAL_DP_INTERFACE    := FALSE,
           MANUAL_MODE              := "DP_VAT".MANUAL_MODE,
           SINGLE_STEP_SLAVE        := "DP_VAT".SINGLE_STEP_SLAVE,
           SINGLE_STEP_ERROR        := "DP_VAT".SINGLE_STEP_ERROR,
           RESET                    := "DP_VAT".RESET,
           SINGLE_DIAG              := "DP_VAT".SINGLE_SLAVE_DIAG,
           SINGLE_DIAG_ADR          := "DP_VAT".SINGLE_DIAG_ADR,
           ALL_DP_SLAVES_OK         := "DP_VAT".ALL_SLAVES_OK,
           SUM_SLAVES_DIAG          := "DP_VAT".SUM_SLAVES_DIAG,
           SLAVE_ADR                := "DP_VAT".SLAVE_ADR,
           SLAVE_STATE              := "DP_VAT".SLAVE_STATE,
           SLAVE_IDENT_NO           := "DP_VAT".SLAVE_IDENT_NO,
           ERROR_NO                 := "DP_VAT".ERROR_NO,
           ERROR_TYPE               := "DP_VAT".ERROR_TYPE,
           MODULE_NO                := "DP_VAT".MODULE_NO,
           MODULE_STATE             := "DP_VAT".MODULE_STATE,
           CHANNEL_NO               := "DP_VAT".CHANNEL_NO,
           CHANNEL_TYPE             := "DP_VAT".CHANNEL_TYPE,
           CHANNEL_ERROR_CODE       := "DP_VAT".CHANNEL_ERROR_CODE,
           CHANNEL_ERROR_INFO_1     := "DP_VAT".CHANNEL_ERROR_INFO_1,
           CHANNEL_ERROR_INFO_2     := "DP_VAT".CHANNEL_ERROR_INFO_2,
           DIAG_COUNTER             := "DP_VAT".DIAG_COUNTER,
           DIAG_OVERFLOW            := "DP_VAT".DIAG_OVERFLOW,
           BUSY                     := "DP_VAT".BUSY);
      NOP   0;
NETWORK
TITLE =
//DP_MASTERSYSTEM=2
      CALL  "DETAIL_DP_DIAG" , "DETAIL_DIAG_DB_RACK1" (
           DP_MASTERSYSTEM          := 2,
           EXTERNAL_DP_INTERFACE    := FALSE,
           MANUAL_MODE              := "DP_VAT".MANUAL_MODE1,
           SINGLE_STEP_SLAVE        := "DP_VAT".SINGLE_STEP_SLAVE1,
           SINGLE_STEP_ERROR        := "DP_VAT".SINGLE_STEP_ERROR1,
           RESET                    := "DP_VAT".RESET1,
           SINGLE_DIAG              := "DP_VAT".SINGLE_SLAVE_DIAG1,
           SINGLE_DIAG_ADR          := "DP_VAT".SINGLE_DIAG_ADR1,
           ALL_DP_SLAVES_OK         := "DP_VAT".ALL_SLAVES_OK1,
           SUM_SLAVES_DIAG          := "DP_VAT".SUM_SLAVES_DIAG1,
           SLAVE_ADR                := "DP_VAT".SLAVE_ADR1,
           SLAVE_STATE              := "DP_VAT".SLAVE_STATE1,
           SLAVE_IDENT_NO           := "DP_VAT".SLAVE_IDENT_NO1,
           ERROR_NO                 := "DP_VAT".ERROR_NO1,
           ERROR_TYPE               := "DP_VAT".ERROR_TYPE1,
           MODULE_NO                := "DP_VAT".MODULE_NO1,
           MODULE_STATE             := "DP_VAT".MODULE_STATE1,
           CHANNEL_NO               := "DP_VAT".CHANNEL_NO1,
           CHANNEL_TYPE             := "DP_VAT".CHANNEL_TYPE1,
           CHANNEL_ERROR_CODE       := "DP_VAT".CHANNEL_ERROR_CODE1,
           CHANNEL_ERROR_INFO_1     := "DP_VAT".CHANNEL_ERROR_INFO_11,
           CHANNEL_ERROR_INFO_2     := "DP_VAT".CHANNEL_ERROR_INFO_21,
           DIAG_COUNTER             := "DP_VAT".DIAG_COUNTER1,
           DIAG_OVERFLOW            := "DP_VAT".DIAG_OVERFLOW1,
           BUSY                     := "DP_VAT".BUSY1);
      NOP   0;
END_ORGANIZATION_BLOCK

ORGANIZATION_BLOCK "COMM_FLT"	// OB 87
TITLE = "Communication Fault"
VERSION : 0.1
VAR_TEMP
  OB87_EV_CLASS : BYTE ;	//16#39 Event class 3
  OB87_FLT_ID : BYTE ;	//16#XX, Fault identifcation code
  OB87_PRIORITY : BYTE ;	//Priority of OB Execution
  OB87_OB_NUMBR : BYTE ;	//87 (Organization block 87, OB87)
  OB87_RESERVED_1 : BYTE ;	//Reserved for system
  OB87_RESERVED_2 : BYTE ;	//Reserved for system
  OB87_RESERVED_3 : WORD ;	//Reserved for system
  OB87_RESERVED_4 : DWORD ;	//Reserved for system
  OB87_DATE_TIME : DATE_AND_TIME ;	//Date and time OB87 started
END_VAR
BEGIN
// (block stored without names or comments; labels and parameter names are numbered)
END_ORGANIZATION_BLOCK

ORGANIZATION_BLOCK "COMPLETE RESTART"	// OB 100
TITLE = "Complete Restart"
VERSION : 0.1
VAR_TEMP
  OB100_EV_CLASS : BYTE ;	//16#13, Event class 1, Entering event state, Event logged in diagnostic buffer
  OB100_STRTUP : BYTE ;	//16#81/82/83/84 Method of startup
  OB100_PRIORITY : BYTE ;	//Priority of OB Execution
  OB100_OB_NUMBR : BYTE ;	//100 (Organization block 100, OB100)
  OB100_RESERVED_1 : BYTE ;	//Reserved for system
  OB100_RESERVED_2 : BYTE ;	//Reserved for system
  OB100_STOP : WORD ;	//Event that caused CPU to stop (16#4xxx)
  OB100_STRT_INFO : DWORD ;	//Information on how system started
  OB100_DATE_TIME : DATE_AND_TIME ;	//Date and time OB100 started
END_VAR
BEGIN
NETWORK
TITLE = Initialisiation of "MB_PNHCL"
//adapt the initialisation parameters according to your configuration
      L     1;
      T     "CONTROL_DAT".id_0_a;
      L     2;
      T     "CONTROL_DAT".id_1_a;
      L     T#5S;
      T     "CONTROL_DAT".reuse_conn_time;
      SET;
      S     "CONTROL_DAT".use_all_conn;
      CALL  "MB_PNHCL" , "IDB_MODBUS" (
           DIW 0                    := "CONTROL_DAT".id_0_a,
           DIW 2                    := "CONTROL_DAT".id_1_a,
           DIW 8                    := 2,
           DID 10                   := "CONTROL_DAT".reuse_conn_time,
           DIX 14.0                 := "CONTROL_DAT".use_all_conn,
           DID 20                   := L#5000,
           DIW 26                   := 3,
           DIX 36.3                 := "CONTROL_DAT".ERROR,
           DIX 36.4                 := "CONTROL_DAT".ESTAB_0A,
           DIW 38                   := "CONTROL_DAT".STATUS_0A,
           DIX 40.0                 := "CONTROL_DAT".ESTAB_1A,
           DIW 42                   := "CONTROL_DAT".STATUS_1A,
           DIX 72.0                 := "CONTROL_DAT".RedErrS7,
           DIX 72.1                 := "CONTROL_DAT".RedErrDev,
           DIX 72.2                 := "CONTROL_DAT".TotComErr);
      A     "CONTROL_DAT".ERROR;
      JCN   end;
      L     "CONTROL_DAT".Count_Error;
      +     1;
      T     "CONTROL_DAT".Count_Error;
      L     "CONTROL_DAT".STATUS_0A;
      T     "CONTROL_DAT".Save_STATUS_0A;
      L     "CONTROL_DAT".STATUS_1A;
      T     "CONTROL_DAT".Save_STATUS_1A;
end:  NOP   0;
END_ORGANIZATION_BLOCK

ORGANIZATION_BLOCK "PROG_ERR"	// OB 121
TITLE = "Programming Error"
VERSION : 0.1
VAR_TEMP
  OB121_EV_CLASS : BYTE ;	//16#25, Event class 2, Entering event state, Internal fault event
  OB121_SW_FLT : BYTE ;	//16#XX Software programming fault
  OB121_PRIORITY : BYTE ;	//Priority of OB Execution
  OB121_OB_NUMBR : BYTE ;	//121 (Organization block 121, OB121)
  OB121_BLK_TYPE : BYTE ;	//16#88/8A/8B/8C/8E Type of block fault occured in
  OB121_RESERVED_1 : BYTE ;	//Reserved for system
  OB121_FLT_REG : WORD ;	//16#XX Specific register that caused fault
  OB121_BLK_NUM : WORD ;	//Number of block that programming fault occured in
  OB121_PRG_ADDR : WORD ;	//Address in block where programming fault occured
  OB121_DATE_TIME : DATE_AND_TIME ;	//Date and time OB121 started
END_VAR
BEGIN
NETWORK
TITLE =
END_ORGANIZATION_BLOCK

ORGANIZATION_BLOCK "MOD_ERR"	// OB 122
TITLE = "Module Access Error"
VERSION : 0.1
VAR_TEMP
  OB122_EV_CLASS : BYTE ;	//16#29, Event class 2, Entering event state, Internal fault event
  OB122_SW_FLT : BYTE ;	//16#XX Software error code
  OB122_PRIORITY : BYTE ;	//Priority of OB Execution
  OB122_OB_NUMBR : BYTE ;	//122 (Organization block 122, OB122)
  OB122_BLK_TYPE : BYTE ;	//16#88/8C/8E Type of block fault occured in
  OB122_MEM_AREA : BYTE ;	//Memory area where access error occured
  OB122_MEM_ADDR : WORD ;	//Memory address where access error occured
  OB122_BLK_NUM : WORD ;	//Block number in which error occured
  OB122_PRG_ADDR : WORD ;	//Program address where error occured
  OB122_DATE_TIME : DATE_AND_TIME ;	//Date and time OB1 started
END_VAR
BEGIN
// (block stored without names or comments; labels and parameter names are numbered)
END_ORGANIZATION_BLOCK

SYMBOL_TABLE
"CPULINDB"	DB 30	DB 30
"FAS1_WR"	DB 2003	DB 2003
"FAS1  RE"	DB 2005	DB 2005
"FAS2_WR"	DB 2013	DB 2013
"FAS2  RE"	DB 2015	DB 2015
"IBP_HMI_SCtrl"	DB 6005	DB 6005
"IBP_ToHMI"	DB 6006	DB 6006
"P_RCV"	FB 12	FB 12	// Receive Data from CP340
"P_SEND"	FB 13	FB 13	// Send Data to CP340
"pid"	FB 41	FB 41
"P_RESET"	FB 177	FB 177	// Reset Job for CP340
"S7400H-COM-MAIN-IBP"	FB 201	FB 201
"IBP-COMM-IBP-MAIN"	FB 203	FB 203
"MODMAS_STEP7_CP340_L"	FB 1071	FB 1071
"HF3_FAS_FB2641"	FB 2641	FB 2641	// FAS主程序
"HF3_FAS_FB2642"	FB 2642	FB 2642
"HF3_FAS_COMM"	FB 2643	FB 2643	// 与FAS通讯功能块
"FAS_MODE_JUDGE"	FB 2644	FB 2644
"AB_IBP_Comm"	FB 2831	FB 2831
"IBP盘与主端通讯"	FB 2833	FB 2833
"HF3_B_T_W_FC51"	FC 51	FC 51	// BOOLתWORD
"HF3_W_T_B_FC54"	FC 54	FC 54	// WORDתBOOL
"GET_DBN"	FC 501	FC 501	// Get DB Nummer
"ZNZM_CURRENT_ILLU_TRANS"	FC 732	FC 732	// 智能低压通信数据段
"HF3_CP340_FC4301"	FC 4301	FC 4301	// CP340_配置程序段
"Always0"	M 0.0	BOOL
"Always1"	M 0.1	BOOL
"RED_I/O_FLT1"	OB 70	OB 70	// Redundancy I/O Fault 1
"RED_FLT"	OB 72	OB 72	// Redundancy Fault
"PS_FLT"	OB 81	OB 81	// Power Supply Fault
"I/O_FLT1"	OB 82	OB 82	// I/O Point Fault 1
"I/O_FLT2"	OB 83	OB 83	// I/O Point Fault 2
"CPU_FLT"	OB 84	OB 84	// CPU Fault
"OBNL_FLT"	OB 85	OB 85	// OB Not Loaded Fault
"RACK_FLT"	OB 86	OB 86	// Loss of Rack Fault
"COMM_FLT"	OB 87	OB 87	// Communication Fault
"COMPLETE RESTART"	OB 100	OB 100	// Complete Restart
"PROG_ERR"	OB 121	OB 121	// Programming Error
"MOD_ERR"	OB 122	OB 122	// Module Access Error
"TON"	SFB 4	SFB 4	// Generate an On Delay
"BSEND"	SFB 12	SFB 12	// Sending Segmented Data
"BRCV"	SFB 13	SFB 13	// Receiving Segmented Data
"RDREC"	SFB 52	SFB 52	// Read a Process Data Record
"WRREC"	SFB 53	SFB 53	// Write a Process Data Record
"TEST_DB"	SFC 24	SFC 24	// Test Data Block
"WR_REC"	SFC 58	SFC 58	// Write Data Record
"RD_REC"	SFC 59	SFC 59	// Read a Data Record
"UDT_ANY_Pointer"	UDT 10	UDT 10
END_SYMBOL_TABLE

TYPE "UDT_ANY_Pointer"	// UDT 10
VERSION : 0.0
  STRUCT
   Syntax_ID : BYTE ;
   DataTyp : BYTE ;
   Count : WORD ;
   DB_Number : WORD ;
   Byte_Pointer : DWORD ;
  END_STRUCT ;	
END_TYPE

// FB 12: know-how protected block, not included

// FB 13: know-how protected block, not included

// FB 41: know-how protected block, not included

// FB 177: know-how protected block, not included

FUNCTION_BLOCK "IBP-COMM-IBP-MAIN"	// FB 203
VERSION : 0.1
VAR_OUTPUT
  STATUS_1 : BOOL ;
  STATUS_2 : BOOL ;
END_VAR
VAR
  BSEND_1 : SFB 12;
  BSEND_2 : SFB 12;
  BREV_1 : SFB 13;
  BREV_2 : SFB 13;
  LENTH : WORD ;
  TON_1 : SFB 4;
  TON_2 : SFB 4;
END_VAR
BEGIN
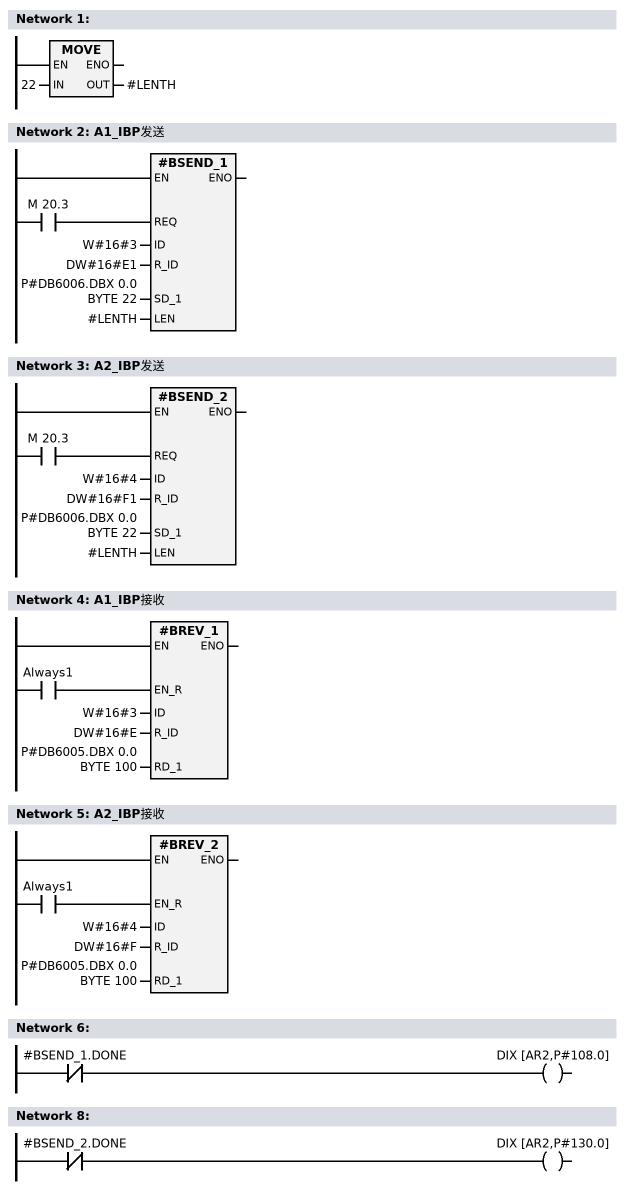
NETWORK
TITLE =
      L     22;
      T     #LENTH;
      NOP   0;
NETWORK
TITLE = A1_IBP发送
      A     M 20.3;
      =     L 0.0;
      BLD   103;
      CALL  #BSEND_1 (
           REQ                      := L 0.0,
           ID                       := W#16#3,
           R_ID                     := DW#16#E1,
           SD_1                     := P#DB6006.DBX 0.0 BYTE 22,
           LEN                      := #LENTH);
      NOP   0;
NETWORK
TITLE = A2_IBP发送
      A     M 20.3;
      =     L 0.0;
      BLD   103;
      CALL  #BSEND_2 (
           REQ                      := L 0.0,
           ID                       := W#16#4,
           R_ID                     := DW#16#F1,
           SD_1                     := P#DB6006.DBX 0.0 BYTE 22,
           LEN                      := #LENTH);
      NOP   0;
NETWORK
TITLE = A1_IBP接收
      A     "Always1";
      =     L 0.0;
      BLD   103;
      CALL  #BREV_1 (
           EN_R                     := L 0.0,
           ID                       := W#16#3,
           R_ID                     := DW#16#E,
           RD_1                     := P#DB6005.DBX 0.0 BYTE 100);
      NOP   0;
NETWORK
TITLE = A2_IBP接收
      A     "Always1";
      =     L 0.0;
      BLD   103;
      CALL  #BREV_2 (
           EN_R                     := L 0.0,
           ID                       := W#16#4,
           R_ID                     := DW#16#F,
           RD_1                     := P#DB6005.DBX 0.0 BYTE 100);
      NOP   0;
NETWORK
TITLE =
      AN    #BSEND_1.DONE;
      =     DIX [AR2,P#108.0];
NETWORK
TITLE =
      BLD   16;
      =     L 7.0;
      L     DINO;
      T     LW 5;
      CDB;
      OPN   DI [LW 5];
      TAR2  LD 1;
      L     L#5000;
      T     DID [AR2,P#110.0];
      +AR2  P#108.0;
      UC    "TON";
      LAR2  LD 1;
      A     DIX [AR2,P#114.0];
      =     DBX [AR2,P#0.0];
      CDB;
      BLD   17;
      NOP   0;
NETWORK
TITLE =
      AN    #BSEND_2.DONE;
      =     DIX [AR2,P#130.0];
NETWORK
TITLE =
      BLD   16;
      =     L 7.0;
      L     DINO;
      T     LW 5;
      CDB;
      OPN   DI [LW 5];
      TAR2  LD 1;
      L     L#5000;
      T     DID [AR2,P#132.0];
      +AR2  P#130.0;
      UC    "TON";
      LAR2  LD 1;
      A     DIX [AR2,P#136.0];
      =     DBX [AR2,P#0.1];
      CDB;
      BLD   17;
      NOP   0;
END_FUNCTION_BLOCK

FUNCTION_BLOCK FB 233
VERSION : 0.0
VAR_OUTPUT
  IBP_A : BOOL ;	//IBP盘自动
  IBP_M : BOOL ;	//IBP盘手动
  EXECUTED_MODE : INT ;	//执行的IBP盘模式号
  RECORD : ARRAY  [0 .. 127 ] OF //对IBP盘面进行的操作记录   //新修改
  BOOL ;	//对IBP盘面进行的操作记录   //新修改
END_VAR
VAR
  Lamp : ARRAY  [0 .. 127 ] OF BOOL ;
  Light : ARRAY  [0 .. 63 ] OF BOOL ;
  i : INT ;
  n : INT ;
  Mode : ARRAY  [0 .. 63 ] OF INT ;
  IBP_AUTO : BOOL ;
  IBP_MANUAL : BOOL ;
END_VAR
BEGIN
// body was compiled from an SCL source; compiled code not shown
END_FUNCTION_BLOCK

// FB 1071: know-how protected block, not included

FUNCTION_BLOCK "HF3_FAS_FB2641"	// FB 2641
VERSION : 0.1
VAR
  FAS : FB 2642;
END_VAR
BEGIN
NETWORK
TITLE =
      BLD   14;
      =     L 6.0;
      L     DINO;
      T     LW 4;
      CDB;
      OPN   DI [LW 4];
      TAR2  LD 0;
      L     2001;
      T     #FAS.FAS1_WORKD_DB;
      L     2011;
      T     #FAS.FAS2_WORKD_DB;
      +AR2  P#0.0;
      UC    "HF3_FAS_FB2642";
      LAR2  LD 0;
      L     #FAS.FAS1_qnWR;
      OPN   DI 2003;
      T     DIW 8;
      OPN   DI [LW 4];
      L     #FAS.FAS2_qnWR;
      OPN   DI 2013;
      T     DIW 8;
      OPN   DI [LW 4];
      L     #FAS.FAS_MODE;
      OPN   DI 6006;
      T     DIW 2;
      OPN   DI [LW 4];
      CDB;
      BLD   15;
      NOP   0;
END_FUNCTION_BLOCK

FUNCTION_BLOCK "HF3_FAS_FB2642"	// FB 2642
VERSION : 0.1
VAR_INPUT
  FAS1_WORKD_DB : INT ;	// FAS主设备work_DB块号
  FAS2_WORKD_DB : INT ;	// FAS备设备work_DB块号
END_VAR
VAR_OUTPUT
  FAS1_qnWR : WORD ;
  FAS2_qnWR : WORD ;
  FAS_MODE : INT ;	// 收到的FAS模式号
  FAS1_CommOK : BOOL ;
  FAS2_CommOK : BOOL ;
END_VAR
VAR
  FAS1 : FB 2643;
  FAS2 : FB 2643;
  JUDGE1 : FB 2644;
  JUDGE2 : FB 2644;
  TON1 : SFB 4;
  TON2 : SFB 4;
  MODE_TEMP1 : INT ;
  MODE_TEMP2 : INT ;
  FAS1_Comm_Statu : BOOL ;
  FAS2_Comm_Statu : BOOL ;
END_VAR
VAR_TEMP
  DB_NO : INT ;
  judge_temp : BOOL ;
END_VAR
BEGIN
NETWORK
TITLE = FAS1  通讯状态判断
      L     #FAS1_WORKD_DB;
      L     4;
      +I;
      T     #DB_NO;
      OPN   DB [#DB_NO];
      L     DBW 2;	//第一条读命令的状态
      L     0;
      <>I;
      =     DIX [AR2,P#464.0];
      BLD   16;
      =     L 9.0;
      L     DINO;
      T     LW 7;
      CDB;
      OPN   DI [LW 7];
      TAR2  LD 3;
      A     DBX [AR2,P#464.0];
      =     DIX [AR2,P#416.0];
      L     L#5000;
      T     DID [AR2,P#418.0];
      +AR2  P#416.0;
      UC    "TON";
      LAR2  LD 3;
      A     DIX [AR2,P#422.0];
      =     #judge_temp;
      CDB;
      BLD   17;
      AN    #judge_temp;
      =     #FAS1_CommOK;
NETWORK
TITLE = FAS2  通讯状态判断
      L     #FAS2_WORKD_DB;
      L     4;
      +I;
      T     #DB_NO;
      OPN   DB [#DB_NO];
      L     DBW 2;	//第一条读命令的状态
      L     0;
      <>I;
      =     DIX [AR2,P#464.1];
      BLD   16;
      =     L 9.0;
      L     DINO;
      T     LW 7;
      CDB;
      OPN   DI [LW 7];
      TAR2  LD 3;
      A     DBX [AR2,P#464.1];
      =     DIX [AR2,P#438.0];
      L     L#5000;
      T     DID [AR2,P#440.0];
      +AR2  P#438.0;
      UC    "TON";
      LAR2  LD 3;
      A     DIX [AR2,P#444.0];
      =     #judge_temp;
      CDB;
      BLD   17;
      AN    #judge_temp;
      =     #FAS2_CommOK;
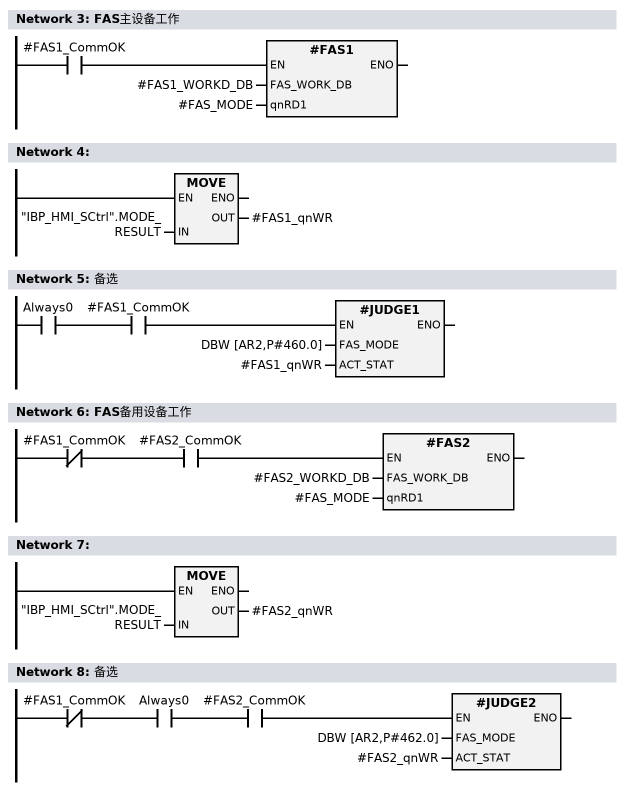
NETWORK
TITLE = FAS主设备工作
      A     #FAS1_CommOK;
      JNB   _001;
      CALL  #FAS1 (
           FAS_WORK_DB              := #FAS1_WORKD_DB,
           qnRD1                    := #FAS_MODE);
_001: NOP   0;
NETWORK
TITLE =
      L     "IBP_HMI_SCtrl".MODE_RESULT;
      T     #FAS1_qnWR;
      NOP   0;
NETWORK
TITLE = 备选
      A     "Always0";
      A     #FAS1_CommOK;
      JNB   _002;
      CALL  #JUDGE1 (
           FAS_MODE                 := DBW [AR2,P#460.0],
           ACT_STAT                 := #FAS1_qnWR);
_002: NOP   0;
NETWORK
TITLE = FAS备用设备工作
      AN    #FAS1_CommOK;
      A     #FAS2_CommOK;
      JNB   _003;
      CALL  #FAS2 (
           FAS_WORK_DB              := #FAS2_WORKD_DB,
           qnRD1                    := #FAS_MODE);
_003: NOP   0;
NETWORK
TITLE =
      L     "IBP_HMI_SCtrl".MODE_RESULT;
      T     #FAS2_qnWR;
      NOP   0;
NETWORK
TITLE = 备选
      AN    #FAS1_CommOK;
      A     "Always0";
      A     #FAS2_CommOK;
      JNB   _004;
      CALL  #JUDGE2 (
           FAS_MODE                 := DBW [AR2,P#462.0],
           ACT_STAT                 := #FAS2_qnWR);
_004: NOP   0;
NETWORK
TITLE =
      SET;
      SAVE;
      CLR;
END_FUNCTION_BLOCK

FUNCTION_BLOCK "HF3_FAS_COMM"	// FB 2643
AUTHOR : SUNWIN_G
FAMILY : FAS
NAME : FAS_CAL
VERSION : 1.1
VAR_INPUT
  FAS_WORK_DB : INT ;	//FASwork_db号
END_VAR
VAR_OUTPUT
  qnRD1 : INT ;	//根据FAS状态点输出模式号
END_VAR
VAR
  FAS_inRD1 : ARRAY  [0 .. 2 ] OF //读取到的FAS状态点
  WORD ;	//读取到的FAS状态点
  FAS_CODE : INT ;	//执行的FAS模式号
  FAS_Encode : ARRAY  [0 .. 47 ] OF //FAS模式号初始化变量
  INT ;	//FAS模式号初始化变量
  i : INT ;
END_VAR
BEGIN
// body was compiled from an SCL source; compiled code not shown
END_FUNCTION_BLOCK

FUNCTION_BLOCK "FAS_MODE_JUDGE"	// FB 2644
VERSION : 0.0
VAR_INPUT
  FAS_MODE : INT ;
  MODE_STATUS : ARRAY  [0 .. 40 ] OF INT ;
END_VAR
VAR_OUTPUT
  ACT_STAT : WORD ;
  STAT : WORD ;
END_VAR
VAR
  system_judge : INT ;	//Static Variables
  system_no : INT ;
END_VAR
BEGIN
// body was compiled from an SCL source; compiled code not shown
END_FUNCTION_BLOCK

FUNCTION_BLOCK "IBP盘与主端通讯"	// FB 2833
VERSION : 0.1
VAR
  IBP_MAIN_COMM : FB 203;
  A1_IBP_CommOK : BOOL ;
  A2_IBP_CommOK : BOOL ;
END_VAR
BEGIN
NETWORK
TITLE = A-IBP通信
      BLD   14;
      =     L 6.0;
      L     DINO;
      T     LW 4;
      CDB;
      OPN   DI [LW 4];
      TAR2  LD 0;
      +AR2  P#0.0;
      UC    "IBP-COMM-IBP-MAIN";
      LAR2  LD 0;
      A     #IBP_MAIN_COMM.STATUS_1;
      =     DBX [AR2,P#152.0];
      A     #IBP_MAIN_COMM.STATUS_2;
      =     DBX [AR2,P#152.1];
      CDB;
      BLD   15;
      NOP   0;
END_FUNCTION_BLOCK

FUNCTION "HF3_B_T_W_FC51" : VOID	// FC 51
VERSION : 0.0
VAR_INPUT
  Bit_0 : BOOL ;
  Bit_1 : BOOL ;
  Bit_2 : BOOL ;
  Bit_3 : BOOL ;
  Bit_4 : BOOL ;
  Bit_5 : BOOL ;
  Bit_6 : BOOL ;
  Bit_7 : BOOL ;
  Bit_8 : BOOL ;
  Bit_9 : BOOL ;
  Bit_10 : BOOL ;
  Bit_11 : BOOL ;
  Bit_12 : BOOL ;
  Bit_13 : BOOL ;
  Bit_14 : BOOL ;
  Bit_15 : BOOL ;
END_VAR
VAR_OUTPUT
  Word1 : WORD ;
END_VAR
VAR_TEMP
  Word2 : WORD ;
END_VAR
BEGIN
// body was compiled from an SCL source; compiled code not shown
END_FUNCTION

FUNCTION "HF3_W_T_B_FC54" : VOID	// FC 54
VERSION : 0.0
VAR_INPUT
  WORD1 : WORD ;
END_VAR
VAR_OUTPUT
  bool1 : ARRAY  [0 .. 15 ] OF
  BOOL ;
END_VAR
BEGIN
NETWORK
TITLE = SCL network
//compiled by SCL compiler version:  SCLCOMP K05.03.07.00_01.02.00.01 release
      SET;
      SAVE;
      =     L 0.1;
      L     #WORD1;
      L     W#16#1;
      AW;
      L     W#16#0;
      <>I;
      BLD   5;
      T     LD 3;
      TAK;
      T     LD 7;
      L     P##bool1;
      LAR1;
      L     W [AR1,P#0.0];
      T     LW 1;
      OPN   DB [LW 1];
      L     D [AR1,P#2.0];
      LAR1;
      L     LD 7;
      L     LD 3;
      =      [AR1,P#0.0];
      L     #WORD1;
      L     W#16#2;
      AW;
      L     W#16#0;
      <>I;
      BLD   5;
      T     LD 3;
      TAK;
      T     LD 7;
      L     P##bool1;
      LAR1;
      L     W [AR1,P#0.0];
      T     LW 1;
      OPN   DB [LW 1];
      L     D [AR1,P#2.0];
      LAR1;
      L     LD 7;
      L     LD 3;
      =      [AR1,P#0.1];
      L     #WORD1;
      L     W#16#4;
      AW;
      L     W#16#0;
      <>I;
      BLD   5;
      T     LD 3;
      TAK;
      T     LD 7;
      L     P##bool1;
      LAR1;
      L     W [AR1,P#0.0];
      T     LW 1;
      OPN   DB [LW 1];
      L     D [AR1,P#2.0];
      LAR1;
      L     LD 7;
      L     LD 3;
      =      [AR1,P#0.2];
      L     #WORD1;
      L     W#16#8;
      AW;
      L     W#16#0;
      <>I;
      BLD   5;
      T     LD 3;
      TAK;
      T     LD 7;
      L     P##bool1;
      LAR1;
      L     W [AR1,P#0.0];
      T     LW 1;
      OPN   DB [LW 1];
      L     D [AR1,P#2.0];
      LAR1;
      L     LD 7;
      L     LD 3;
      =      [AR1,P#0.3];
      L     #WORD1;
      L     W#16#10;
      AW;
      L     W#16#0;
      <>I;
      BLD   5;
      T     LD 3;
      TAK;
      T     LD 7;
      L     P##bool1;
      LAR1;
      L     W [AR1,P#0.0];
      T     LW 1;
      OPN   DB [LW 1];
      L     D [AR1,P#2.0];
      LAR1;
      L     LD 7;
      L     LD 3;
      =      [AR1,P#0.4];
      L     #WORD1;
      L     W#16#20;
      AW;
      L     W#16#0;
      <>I;
      BLD   5;
      T     LD 3;
      TAK;
      T     LD 7;
      L     P##bool1;
      LAR1;
      L     W [AR1,P#0.0];
      T     LW 1;
      OPN   DB [LW 1];
      L     D [AR1,P#2.0];
      LAR1;
      L     LD 7;
      L     LD 3;
      =      [AR1,P#0.5];
      L     #WORD1;
      L     W#16#40;
      AW;
      L     W#16#0;
      <>I;
      BLD   5;
      T     LD 3;
      TAK;
      T     LD 7;
      L     P##bool1;
      LAR1;
      L     W [AR1,P#0.0];
      T     LW 1;
      OPN   DB [LW 1];
      L     D [AR1,P#2.0];
      LAR1;
      L     LD 7;
      L     LD 3;
      =      [AR1,P#0.6];
      L     #WORD1;
      L     W#16#80;
      AW;
      L     W#16#0;
      <>I;
      BLD   5;
      T     LD 3;
      TAK;
      T     LD 7;
      L     P##bool1;
      LAR1;
      L     W [AR1,P#0.0];
      T     LW 1;
      OPN   DB [LW 1];
      L     D [AR1,P#2.0];
      LAR1;
      L     LD 7;
      L     LD 3;
      =      [AR1,P#0.7];
      L     #WORD1;
      L     W#16#100;
      AW;
      L     W#16#0;
      <>I;
      BLD   5;
      T     LD 3;
      TAK;
      T     LD 7;
      L     P##bool1;
      LAR1;
      L     W [AR1,P#0.0];
      T     LW 1;
      OPN   DB [LW 1];
      L     D [AR1,P#2.0];
      LAR1;
      L     LD 7;
      L     LD 3;
      =      [AR1,P#1.0];
      L     #WORD1;
      L     W#16#200;
      AW;
      L     W#16#0;
      <>I;
      BLD   5;
      T     LD 3;
      TAK;
      T     LD 7;
      L     P##bool1;
      LAR1;
      L     W [AR1,P#0.0];
      T     LW 1;
      OPN   DB [LW 1];
      L     D [AR1,P#2.0];
      LAR1;
      L     LD 7;
      L     LD 3;
      =      [AR1,P#1.1];
      L     #WORD1;
      L     W#16#400;
      AW;
      L     W#16#0;
      <>I;
      BLD   5;
      T     LD 3;
      TAK;
      T     LD 7;
      L     P##bool1;
      LAR1;
      L     W [AR1,P#0.0];
      T     LW 1;
      OPN   DB [LW 1];
      L     D [AR1,P#2.0];
      LAR1;
      L     LD 7;
      L     LD 3;
      =      [AR1,P#1.2];
      L     #WORD1;
      L     W#16#800;
      AW;
      L     W#16#0;
      <>I;
      BLD   5;
      T     LD 3;
      TAK;
      T     LD 7;
      L     P##bool1;
      LAR1;
      L     W [AR1,P#0.0];
      T     LW 1;
      OPN   DB [LW 1];
      L     D [AR1,P#2.0];
      LAR1;
      L     LD 7;
      L     LD 3;
      =      [AR1,P#1.3];
      L     #WORD1;
      L     W#16#1000;
      AW;
      L     W#16#0;
      <>I;
      BLD   5;
      T     LD 3;
      TAK;
      T     LD 7;
      L     P##bool1;
      LAR1;
      L     W [AR1,P#0.0];
      T     LW 1;
      OPN   DB [LW 1];
      L     D [AR1,P#2.0];
      LAR1;
      L     LD 7;
      L     LD 3;
      =      [AR1,P#1.4];
      L     #WORD1;
      L     W#16#2000;
      AW;
      L     W#16#0;
      <>I;
      BLD   5;
      T     LD 3;
      TAK;
      T     LD 7;
      L     P##bool1;
      LAR1;
      L     W [AR1,P#0.0];
      T     LW 1;
      OPN   DB [LW 1];
      L     D [AR1,P#2.0];
      LAR1;
      L     LD 7;
      L     LD 3;
      =      [AR1,P#1.5];
      L     #WORD1;
      L     W#16#4000;
      AW;
      L     W#16#0;
      <>I;
      BLD   5;
      T     LD 3;
      TAK;
      T     LD 7;
      L     P##bool1;
      LAR1;
      L     W [AR1,P#0.0];
      T     LW 1;
      OPN   DB [LW 1];
      L     D [AR1,P#2.0];
      LAR1;
      L     LD 7;
      L     LD 3;
      =      [AR1,P#1.6];
      L     #WORD1;
      L     W#16#8000;
      AW;
      L     W#16#0;
      <>I;
      BLD   5;
      T     LD 3;
      TAK;
      T     LD 7;
      L     P##bool1;
      LAR1;
      L     W [AR1,P#0.0];
      T     LW 1;
      OPN   DB [LW 1];
      L     D [AR1,P#2.0];
      LAR1;
      L     LD 7;
      L     LD 3;
      =      [AR1,P#1.7];
      A     L 0.1;
      SAVE;
      BE;
END_FUNCTION

// FC 501: know-how protected block, not included

FUNCTION "ZNZM_CURRENT_ILLU_TRANS" : VOID	// FC 732
VERSION : 0.1
VAR_INPUT
  in_Lux : WORD ;
END_VAR
VAR_OUTPUT
  lux_Real : REAL ;
END_VAR
VAR_TEMP
  temp1 : INT ;
  temp2 : INT ;
  temp3 : INT ;
  temp4 : INT ;
  temp5 : INT ;
  temp6 : INT ;
  temp7 : INT ;
  temp8 : INT ;
  end : BOOL ;
  BOOl_array : ARRAY  [0 .. 15 ] OF BOOL ;
  M : WORD ;
  E : WORD ;
  M_INT : INT ;
  E_INT : INT ;
  M_OUT : INT ;
END_VAR
BEGIN
NETWORK
TITLE =
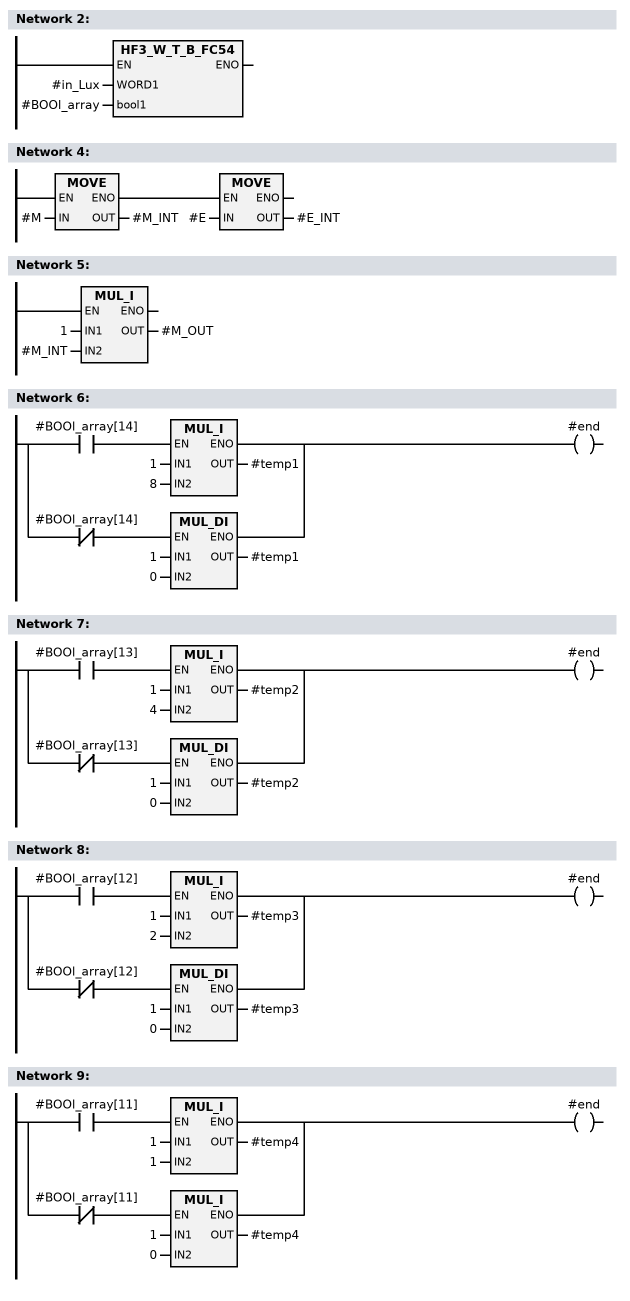
NETWORK
TITLE =
      CALL  "HF3_W_T_B_FC54" (
           WORD1                    := #in_Lux,
           bool1                    := #BOOl_array);
      NOP   0;
NETWORK
TITLE =
      A     #BOOl_array[11];
      =     L 30.0;
      BLD   103;
      A     #BOOl_array[12];
      =     L 30.1;
      BLD   103;
      A     #BOOl_array[13];
      =     L 30.2;
      BLD   103;
      A     #BOOl_array[14];
      =     L 30.3;
      BLD   103;
      A     "Always0";
      =     L 30.4;
      BLD   103;
      A     "Always0";
      =     L 30.5;
      BLD   103;
      A     "Always0";
      =     L 30.6;
      BLD   103;
      A     "Always0";
      =     L 30.7;
      BLD   103;
      A     "Always0";
      =     L 31.0;
      BLD   103;
      A     "Always0";
      =     L 31.1;
      BLD   103;
      A     "Always0";
      =     L 31.2;
      BLD   103;
      A     "Always0";
      =     L 31.3;
      BLD   103;
      A     "Always0";
      =     L 31.4;
      BLD   103;
      A     "Always0";
      =     L 31.5;
      BLD   103;
      A     "Always0";
      =     L 31.6;
      BLD   103;
      A     "Always0";
      =     L 31.7;
      BLD   103;
      A(;
      A     #BOOl_array[0];
      =     L 32.0;
      BLD   103;
      A     #BOOl_array[1];
      =     L 32.1;
      BLD   103;
      A     #BOOl_array[2];
      =     L 32.2;
      BLD   103;
      A     #BOOl_array[3];
      =     L 32.3;
      BLD   103;
      A     #BOOl_array[4];
      =     L 32.4;
      BLD   103;
      A     #BOOl_array[5];
      =     L 32.5;
      BLD   103;
      A     #BOOl_array[6];
      =     L 32.6;
      BLD   103;
      A     #BOOl_array[7];
      =     L 32.7;
      BLD   103;
      A     #BOOl_array[8];
      =     L 33.0;
      BLD   103;
      A     #BOOl_array[9];
      =     L 33.1;
      BLD   103;
      A     #BOOl_array[10];
      =     L 33.2;
      BLD   103;
      A     #BOOl_array[15];
      =     L 33.3;
      BLD   103;
      A     "Always0";
      =     L 33.4;
      BLD   103;
      A     "Always0";
      =     L 33.5;
      BLD   103;
      A     "Always0";
      =     L 33.6;
      BLD   103;
      A     "Always0";
      =     L 33.7;
      BLD   103;
      CALL  "HF3_B_T_W_FC51" (
           Bit_0                    := L 32.0,
           Bit_1                    := L 32.1,
           Bit_2                    := L 32.2,
           Bit_3                    := L 32.3,
           Bit_4                    := L 32.4,
           Bit_5                    := L 32.5,
           Bit_6                    := L 32.6,
           Bit_7                    := L 32.7,
           Bit_8                    := L 33.0,
           Bit_9                    := L 33.1,
           Bit_10                   := L 33.2,
           Bit_11                   := L 33.3,
           Bit_12                   := L 33.4,
           Bit_13                   := L 33.5,
           Bit_14                   := L 33.6,
           Bit_15                   := L 33.7,
           Word1                    := #M);
      A     BR;
      );
      JNB   _001;
      CALL  "HF3_B_T_W_FC51" (
           Bit_0                    := L 30.0,
           Bit_1                    := L 30.1,
           Bit_2                    := L 30.2,
           Bit_3                    := L 30.3,
           Bit_4                    := L 30.4,
           Bit_5                    := L 30.5,
           Bit_6                    := L 30.6,
           Bit_7                    := L 30.7,
           Bit_8                    := L 31.0,
           Bit_9                    := L 31.1,
           Bit_10                   := L 31.2,
           Bit_11                   := L 31.3,
           Bit_12                   := L 31.4,
           Bit_13                   := L 31.5,
           Bit_14                   := L 31.6,
           Bit_15                   := L 31.7,
           Word1                    := #E);
_001: NOP   0;
NETWORK
TITLE =
      A(;
      L     #M;
      T     #M_INT;
      SET;
      SAVE;
      CLR;
      A     BR;
      );
      JNB   _002;
      L     #E;
      T     #E_INT;
_002: NOP   0;
NETWORK
TITLE =
      L     1;
      L     #M_INT;
      *I;
      T     #M_OUT;
      NOP   0;
NETWORK
TITLE =
      O(;
      A     #BOOl_array[14];
      JNB   _003;
      L     1;
      L     8;
      *I;
      T     #temp1;
      AN    OV;
      SAVE;
      CLR;
_003: A     BR;
      );
      O(;
      AN    #BOOl_array[14];
      JNB   _004;
      L     1;
      L     0;
      *D;
      T     #temp1;
      AN    OV;
      SAVE;
      CLR;
_004: A     BR;
      );
      =     #end;
NETWORK
TITLE =
      O(;
      A     #BOOl_array[13];
      JNB   _005;
      L     1;
      L     4;
      *I;
      T     #temp2;
      AN    OV;
      SAVE;
      CLR;
_005: A     BR;
      );
      O(;
      AN    #BOOl_array[13];
      JNB   _006;
      L     1;
      L     0;
      *D;
      T     #temp2;
      AN    OV;
      SAVE;
      CLR;
_006: A     BR;
      );
      =     #end;
NETWORK
TITLE =
      O(;
      A     #BOOl_array[12];
      JNB   _007;
      L     1;
      L     2;
      *I;
      T     #temp3;
      AN    OV;
      SAVE;
      CLR;
_007: A     BR;
      );
      O(;
      AN    #BOOl_array[12];
      JNB   _008;
      L     1;
      L     0;
      *D;
      T     #temp3;
      AN    OV;
      SAVE;
      CLR;
_008: A     BR;
      );
      =     #end;
NETWORK
TITLE =
      O(;
      A     #BOOl_array[11];
      JNB   _009;
      L     1;
      L     1;
      *I;
      T     #temp4;
      AN    OV;
      SAVE;
      CLR;
_009: A     BR;
      );
      O(;
      AN    #BOOl_array[11];
      JNB   _00a;
      L     1;
      L     0;
      *I;
      T     #temp4;
      AN    OV;
      SAVE;
      CLR;
_00a: A     BR;
      );
      =     #end;
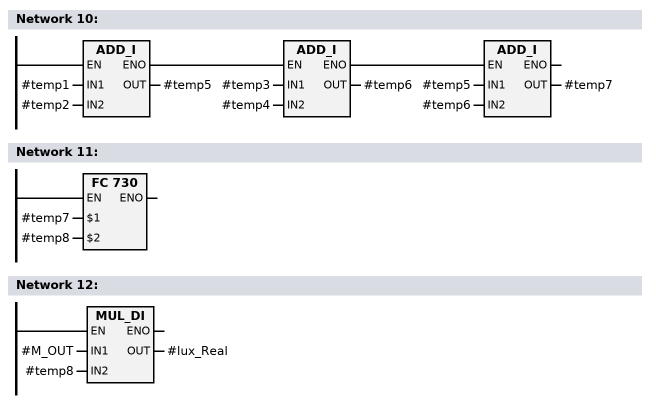
NETWORK
TITLE =
      A(;
      A(;
      L     #temp1;
      L     #temp2;
      +I;
      T     #temp5;
      AN    OV;
      SAVE;
      CLR;
      A     BR;
      );
      JNB   _00b;
      L     #temp3;
      L     #temp4;
      +I;
      T     #temp6;
      AN    OV;
      SAVE;
      CLR;
_00b: A     BR;
      );
      JNB   _00c;
      L     #temp5;
      L     #temp6;
      +I;
      T     #temp7;
_00c: NOP   0;
NETWORK
TITLE =
      CALL  FC 730 (
           $1                       := #temp7,
           $2                       := #temp8);
      NOP   0;
NETWORK
TITLE =
      L     #M_OUT;
      L     #temp8;
      *D;
      T     #lux_Real;
      NOP   0;
END_FUNCTION

FUNCTION "HF3_CP340_FC4301" : VOID	// FC 4301
TITLE = 配置本端所有CP340模块
//1：硬件配置 设置协议、波特率、奇偶校验位、起始地址
//2：需授权
//3：注意起始地址、DB块号（暂未填写）
VERSION : 0.1
BEGIN
NETWORK
TITLE = FAS1 512 2001~2005
      A     "Always0";
      =     L 0.0;
      BLD   103;
      A     "Always1";
      =     L 0.1;
      BLD   103;
      BLD   3;
      =     L 5.0;
      CDB;
      OPN   DI 1071;
      TAR2  LD 1;
      L     512;
      T     DIW 0;
      A     L 0.0;
      =     DIX 4.0;
      L     B#16#4A;
      T     DIB 5;
      L     31001;
      T     DIW 6;
      L     5;
      T     DIW 8;
      L     L#500;
      T     DID 10;
      A     L 0.1;
      =     DIX 14.0;
      L     2001;
      T     DIW 16;
      BLD   11;
      L     W#16#1002;
      T     LW 8;
      L     10;
      T     LW 10;
      L     30;
      T     LW 12;
      L     P#DBX 0.0;
      T     LD 14;
      L     W#16#1002;
      T     LW 18;
      L     10;
      T     LW 20;
      L     1071;
      T     LW 22;
      L     P#DBX 18.0;
      T     LD 24;
      UC    SFC 20;
      {     P#L 8.0, P#L 6.0, P#L 18.0 };
      LAR2  P#DBX 0.0;
      UC    "MODMAS_STEP7_CP340_L";
      LAR2  LD 1;
      A     DIX 38.0;
      =     M 10.0;
      L     DIW 40;
      T     MW 12;
      L     DIW 42;
      T     MW 14;
      CDB;
      BLD   4;
      NOP   0;
NETWORK
TITLE = FAS2  528 2011~2015
      A     "Always0";
      =     L 0.0;
      BLD   103;
      A     "Always1";
      =     L 0.1;
      BLD   103;
      BLD   3;
      =     L 5.0;
      CDB;
      OPN   DI 1072;
      TAR2  LD 1;
      L     528;
      T     DIW 0;
      A     L 0.0;
      =     DIX 4.0;
      L     B#16#4A;
      T     DIB 5;
      L     31001;
      T     DIW 6;
      L     5;
      T     DIW 8;
      L     L#500;
      T     DID 10;
      A     L 0.1;
      =     DIX 14.0;
      L     2011;
      T     DIW 16;
      BLD   11;
      L     W#16#1002;
      T     LW 8;
      L     10;
      T     LW 10;
      L     30;
      T     LW 12;
      L     P#DBX 0.0;
      T     LD 14;
      L     W#16#1002;
      T     LW 18;
      L     10;
      T     LW 20;
      L     1072;
      T     LW 22;
      L     P#DBX 18.0;
      T     LD 24;
      UC    SFC 20;
      {     P#L 8.0, P#L 6.0, P#L 18.0 };
      LAR2  P#DBX 0.0;
      UC    "MODMAS_STEP7_CP340_L";
      LAR2  LD 1;
      A     DIX 38.0;
      =     M 10.0;
      L     DIW 40;
      T     MW 12;
      L     DIW 42;
      T     MW 14;
      CDB;
      BLD   4;
      NOP   0;
END_FUNCTION

DATA_BLOCK "CPULINDB"	// DB 30
VERSION : 0.1
  STRUCT
   YOULIN1 : STRING  [8 ] := 'P5H7L9P4';	//Temporary placeholder variable
   YOULIN2 : STRING  [8 ];
  END_STRUCT ;	
BEGIN
   YOULIN1 := 'P5H7L9P4';
END_DATA_BLOCK

DATA_BLOCK DB 233
VERSION : 0.0
FB 233
BEGIN
END_DATA_BLOCK

DATA_BLOCK DB 234
//
// Block Comment ...
//
//
VERSION : 0.0
  STRUCT
   RECORD_ARCHIVED : INT ;	//传给综合监控的操作记录
  END_STRUCT ;	
BEGIN
END_DATA_BLOCK

DATA_BLOCK DB 1000
VERSION : 0.0
"IBP盘与主端通讯"
BEGIN
END_DATA_BLOCK

DATA_BLOCK DB 1071
AUTHOR : Dixinke
FAMILY : ASCMOD
VERSION : 0.0
"MODMAS_STEP7_CP340_L"
BEGIN
END_DATA_BLOCK

DATA_BLOCK DB 1072
AUTHOR : Dixinke
FAMILY : ASCMOD
VERSION : 0.0
"MODMAS_STEP7_CP340_L"
BEGIN
END_DATA_BLOCK

DATA_BLOCK DB 2001
VERSION : 0.0
  STRUCT
   START_SEQ : BYTE  := B#16#1;
   END_SEQ : BYTE  := B#16#2;
   SND_COMM_DB : WORD  := W#16#7D2;
   WRT_COMM_DB : WORD  := W#16#7D3;
   WRT_COMP_DB : WORD  := W#16#7D4;
   DAT_RECV_DB : WORD  := W#16#7D5;
   ACT_1 : BOOL  := TRUE;
   Mode_1 : BOOL ;
   SND_DB_1 : INT  := 2004;
   SND_ADD_1 : INT ;
   SND_LEN_1 : INT  := 10;
   RCV_DB_1 : INT  := 2005;
   RCV_ADD_1 : INT ;
   RCV_LEN_1 : INT  := 2;
   WD_TIME_1 : INT  := 3000;
   ACT_2 : BOOL  := TRUE;
   Mode_2 : BOOL ;
   SND_DB_2 : INT  := 2002;
   SND_ADD_2 : INT ;
   SND_LEN_2 : INT  := 6;
   RCV_DB_2 : INT  := 2005;
   RCV_ADD_2 : INT  := 2;
   RCV_LEN_2 : INT  := 8;
   WD_TIME_2 : INT  := 3000;
  END_STRUCT ;	
BEGIN
   START_SEQ := B#16#1;
   END_SEQ := B#16#2;
   SND_COMM_DB := W#16#7D2;
   WRT_COMM_DB := W#16#7D3;
   WRT_COMP_DB := W#16#7D4;
   DAT_RECV_DB := W#16#7D5;
   ACT_1 := TRUE;
   SND_DB_1 := 2004;
   SND_LEN_1 := 10;
   RCV_DB_1 := 2005;
   RCV_LEN_1 := 2;
   WD_TIME_1 := 3000;
   ACT_2 := TRUE;
   SND_DB_2 := 2002;
   SND_LEN_2 := 6;
   RCV_DB_2 := 2005;
   RCV_ADD_2 := 2;
   RCV_LEN_2 := 8;
   WD_TIME_2 := 3000;
END_DATA_BLOCK

DATA_BLOCK DB 2002
VERSION : 0.0
  STRUCT
   SlaveID_2 : BYTE  := B#16#B;
   FC_2 : BYTE  := B#16#3;
   START_ADD_2 : WORD  := W#16#1;
   DATA_NUM_2 : WORD  := W#16#3;
   CRC_2 : WORD ;
  END_STRUCT ;	
BEGIN
   SlaveID_2 := B#16#B;
   FC_2 := B#16#3;
   START_ADD_2 := W#16#1;
   DATA_NUM_2 := W#16#3;
END_DATA_BLOCK

DATA_BLOCK "FAS1_WR"	// DB 2003
VERSION : 0.0
  STRUCT
   SlaveID_1 : BYTE  := B#16#B;
   FC_1 : BYTE  := B#16#10;
   START_ADD_1 : WORD ;
   DATA_NUM_1 : WORD  := W#16#1;
   DATA_BYTE_1 : WORD  := W#16#2;
   DATA_1_1 : WORD ;	//地址40001
   CRC_1 : WORD ;
  END_STRUCT ;	
BEGIN
   SlaveID_1 := B#16#B;
   FC_1 := B#16#10;
   DATA_NUM_1 := W#16#1;
   DATA_BYTE_1 := W#16#2;
END_DATA_BLOCK

DATA_BLOCK DB 2004
VERSION : 0.0
  STRUCT
   SlaveID_1 : BYTE  := B#16#B;
   FC_1 : BYTE  := B#16#10;
   START_ADD_1 : WORD ;
   DATA_NUM_1 : WORD  := W#16#1;
   DATA_BYTE_1 : WORD  := W#16#2;
   DATA_NUM_1_1 : WORD ;
   CRC_1 : WORD ;
  END_STRUCT ;	
BEGIN
   SlaveID_1 := B#16#B;
   FC_1 := B#16#10;
   DATA_NUM_1 := W#16#1;
   DATA_BYTE_1 := W#16#2;
END_DATA_BLOCK

DATA_BLOCK "FAS1  RE"	// DB 2005
VERSION : 0.0
  STRUCT
   Command_1_STATUS : WORD ;	//第1条命令的状态，0=正常，1=无响应，2=站号错误，3=命令错误，4=CRC校验错误
   Command_2_STATUS : WORD ;	//第2条命令的状态，0=正常，1=无响应，2=站号错误，3=命令错误，4=CRC校验错误
   Command_2_DATA_1 : WORD ;	//地址40002
   Command_2_DATA_2 : WORD ;	//地址40003
   Command_2_DATA_3 : WORD ;	//地址40004
  END_STRUCT ;	
BEGIN
END_DATA_BLOCK

DATA_BLOCK DB 2011
VERSION : 0.0
  STRUCT
   START_SEQ : BYTE  := B#16#1;
   END_SEQ : BYTE  := B#16#2;
   SND_COMM_DB : WORD  := W#16#7DC;
   WRT_COMM_DB : WORD  := W#16#7DD;
   WRT_COMP_DB : WORD  := W#16#7DE;
   DAT_RECV_DB : WORD  := W#16#7DF;
   ACT_1 : BOOL  := TRUE;
   Mode_1 : BOOL ;
   SND_DB_1 : INT  := 2014;
   SND_ADD_1 : INT ;
   SND_LEN_1 : INT  := 10;
   RCV_DB_1 : INT  := 2015;
   RCV_ADD_1 : INT ;
   RCV_LEN_1 : INT  := 2;
   WD_TIME_1 : INT  := 3000;
   ACT_2 : BOOL  := TRUE;
   Mode_2 : BOOL ;
   SND_DB_2 : INT  := 2012;
   SND_ADD_2 : INT ;
   SND_LEN_2 : INT  := 6;
   RCV_DB_2 : INT  := 2015;
   RCV_ADD_2 : INT  := 2;
   RCV_LEN_2 : INT  := 8;
   WD_TIME_2 : INT  := 3000;
  END_STRUCT ;	
BEGIN
   START_SEQ := B#16#1;
   END_SEQ := B#16#2;
   SND_COMM_DB := W#16#7DC;
   WRT_COMM_DB := W#16#7DD;
   WRT_COMP_DB := W#16#7DE;
   DAT_RECV_DB := W#16#7DF;
   ACT_1 := TRUE;
   SND_DB_1 := 2014;
   SND_LEN_1 := 10;
   RCV_DB_1 := 2015;
   RCV_LEN_1 := 2;
   WD_TIME_1 := 3000;
   ACT_2 := TRUE;
   SND_DB_2 := 2012;
   SND_LEN_2 := 6;
   RCV_DB_2 := 2015;
   RCV_ADD_2 := 2;
   RCV_LEN_2 := 8;
   WD_TIME_2 := 3000;
END_DATA_BLOCK

DATA_BLOCK DB 2012
VERSION : 0.0
  STRUCT
   SlaveID_2 : BYTE  := B#16#C;
   FC_2 : BYTE  := B#16#3;
   START_ADD_2 : WORD  := W#16#1;
   DATA_NUM_2 : WORD  := W#16#3;
   CRC_2 : WORD ;
  END_STRUCT ;	
BEGIN
   SlaveID_2 := B#16#C;
   FC_2 := B#16#3;
   START_ADD_2 := W#16#1;
   DATA_NUM_2 := W#16#3;
END_DATA_BLOCK

DATA_BLOCK "FAS2_WR"	// DB 2013
VERSION : 0.0
  STRUCT
   SlaveID_1 : BYTE  := B#16#C;
   FC_1 : BYTE  := B#16#10;
   START_ADD_1 : WORD ;
   DATA_NUM_1 : WORD  := W#16#1;
   DATA_BYTE_1 : WORD  := W#16#2;
   DATA_1_1 : WORD ;	//地址40001
   CRC_1 : WORD ;
  END_STRUCT ;	
BEGIN
   SlaveID_1 := B#16#C;
   FC_1 := B#16#10;
   DATA_NUM_1 := W#16#1;
   DATA_BYTE_1 := W#16#2;
END_DATA_BLOCK

DATA_BLOCK DB 2014
VERSION : 0.0
  STRUCT
   SlaveID_1 : BYTE  := B#16#C;
   FC_1 : BYTE  := B#16#10;
   START_ADD_1 : WORD ;
   DATA_NUM_1 : WORD  := W#16#1;
   DATA_BYTE_1 : WORD  := W#16#2;
   DATA_NUM_1_1 : WORD ;
   CRC_1 : WORD ;
  END_STRUCT ;	
BEGIN
   SlaveID_1 := B#16#C;
   FC_1 := B#16#10;
   DATA_NUM_1 := W#16#1;
   DATA_BYTE_1 := W#16#2;
END_DATA_BLOCK

DATA_BLOCK "FAS2  RE"	// DB 2015
VERSION : 0.0
  STRUCT
   Command_1_STATUS : WORD ;	//第1条命令的状态，0=正常，1=无响应，2=站号错误，3=命令错误，4=CRC校验错误
   Command_2_STATUS : WORD ;	//第2条命令的状态，0=正常，1=无响应，2=站号错误，3=命令错误，4=CRC校验错误
   Command_2_DATA_1 : WORD ;	//地址40002
   Command_2_DATA_2 : WORD ;	//地址40003
   Command_2_DATA_3 : WORD ;	//地址40004
  END_STRUCT ;	
BEGIN
END_DATA_BLOCK

DATA_BLOCK DB 3202
VERSION : 0.0
"HF3_FAS_FB2641"
BEGIN
END_DATA_BLOCK

DATA_BLOCK "IBP_HMI_SCtrl"	// DB 6005
VERSION : 0.1
  STRUCT
   ActSTAT : ARRAY  [0 .. 40 ] OF //Temporary placeholder variable
   INT  := 0;
   MODE_RESULT : INT ;	//火灾模式执行结果
   reserved : ARRAY  [0 .. 7 ] OF INT ;
  END_STRUCT ;	
BEGIN
END_DATA_BLOCK

DATA_BLOCK "IBP_ToHMI"	// DB 6006
VERSION : 0.0
  STRUCT
   IBP_Mode_Num : INT ;	//执行模式号
   FAS_CODE : INT ;	//FAS火灾模式号
   IBP_Auto : BOOL ;	//自动
   IBP_Manual : BOOL ;	//手动
   IBP_Record : ARRAY  [0 .. 127 ] OF //操作记录
   BOOL  := FALSE;
  END_STRUCT ;	
BEGIN
   IBP_Mode_Num := 1142;
END_DATA_BLOCK

ORGANIZATION_BLOCK OB 1
TITLE = "Main Program Sweep (Cycle)"
VERSION : 0.1
VAR_TEMP
  OB1_EV_CLASS : BYTE ;	//Bits 0-3 = 1 (Coming event), Bits 4-7 = 1 (Event class 1)
  OB1_SCAN_1 : BYTE ;	//1 (Cold restart scan 1 of OB 1), 3 (Scan 2-n of OB 1)
  OB1_PRIORITY : BYTE ;	//Priority of OB Execution
  OB1_OB_NUMBR : BYTE ;	//1 (Organization block 1, OB1)
  OB1_RESERVED_1 : BYTE ;	//Reserved for system
  OB1_RESERVED_2 : BYTE ;	//Reserved for system
  OB1_PREV_CYCLE : INT ;	//Cycle time of previous OB1 scan (milliseconds)
  OB1_MIN_CYCLE : INT ;	//Minimum cycle time of OB1 (milliseconds)
  OB1_MAX_CYCLE : INT ;	//Maximum cycle time of OB1 (milliseconds)
  OB1_DATE_TIME : DATE_AND_TIME ;	//Date and time OB1 started
END_VAR
BEGIN
NETWORK
TITLE = IBP盘手动模式处理
// (network holds code this reader does not know; not shown)
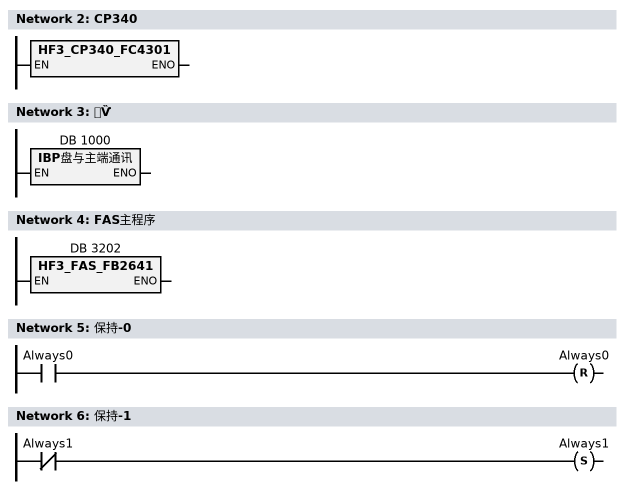
NETWORK
TITLE = CP340
      CALL  "HF3_CP340_FC4301";
      NOP   0;
NETWORK
TITLE = ͨѶ
      CALL  "IBP盘与主端通讯" , DB 1000;
      NOP   0;
NETWORK
TITLE = FAS主程序
      CALL  "HF3_FAS_FB2641" , DB 3202;
      NOP   0;
NETWORK
TITLE = 保持-0
      A     "Always0";
      R     "Always0";
NETWORK
TITLE = 保持-1
      AN    "Always1";
      S     "Always1";
END_ORGANIZATION_BLOCK

ORGANIZATION_BLOCK "RED_I/O_FLT1"	// OB 70
TITLE = "Redundancy I/O Fault 1"
VERSION : 0.1
VAR_TEMP
  OB70_EV_CLASS : BYTE ;	//Event class 7, module inserted/removed (8/9)
  OB70_FLT_ID : BYTE ;	//Fault identifcation code
  OB70_PRIORITY : BYTE ;	//Priority of OB Execution
  OB70_OB_NUMBR : BYTE ;	//70 (Organization block 70, OB70)
  OB70_RESERVED_1 : WORD ;	//Reserved for system
  OB70_INFO_1 : WORD ;	//Info 1
  OB70_INFO_2 : WORD ;	//Info 2
  OB70_INFO_3 : WORD ;	//Info 3
  OB70_DATE_TIME : DATE_AND_TIME ;	//Date and time OB70 started
END_VAR
BEGIN
// (block stored without names or comments; labels and parameter names are numbered)
END_ORGANIZATION_BLOCK

ORGANIZATION_BLOCK "RED_FLT"	// OB 72
TITLE = "Redundancy Fault"
VERSION : 0.1
VAR_TEMP
  OB72_EV_CLASS : BYTE ;	//Event class 7, module inserted/removed (8/9)
  OB72_FLT_ID : BYTE ;	//Fault identifcation code
  OB72_PRIORITY : BYTE ;	//Priority of OB Execution
  OB72_OB_NUMBR : BYTE ;	//72 (Organization block 72, OB72)
  OB72_RESERVED_1 : WORD ;	//Reserved for system
  OB72_INFO_1 : WORD ;	//Info 1
  OB72_INFO_2 : WORD ;	//Info 2
  OB72_INFO_3 : WORD ;	//Info 3
  OB72_DATE_TIME : DATE_AND_TIME ;	//Date and time OB72 started
END_VAR
BEGIN
// (block stored without names or comments; labels and parameter names are numbered)
END_ORGANIZATION_BLOCK

ORGANIZATION_BLOCK "PS_FLT"	// OB 81
TITLE = "Power Supply Fault"
VERSION : 0.1
VAR_TEMP
  OB81_EV_CLASS : BYTE ;	//16#39, Event class 3, Entering event state, Internal fault event
  OB81_FLT_ID : BYTE ;	//16#XX, Fault identifcation code
  OB81_PRIORITY : BYTE ;	//Priority of OB Execution
  OB81_OB_NUMBR : BYTE ;	//81 (Organization block 81, OB81)
  OB81_RESERVED_1 : BYTE ;	//Reserved for system
  OB81_RESERVED_2 : BYTE ;	//Reserved for system
  OB81_RACK_CPU : WORD ;	//see online help (F1)
  OB81_RESERVED_3 : BYTE ;	//Reserved for system
  OB81_RESERVED_4 : BYTE ;	//Reserved for system
  OB81_RESERVED_5 : BYTE ;	//Reserved for system
  OB81_RESERVED_6 : BYTE ;	//Reserved for system
  OB81_DATE_TIME : DATE_AND_TIME ;	//Date and time OB81 started
END_VAR
BEGIN
// (block stored without names or comments; labels and parameter names are numbered)
END_ORGANIZATION_BLOCK

ORGANIZATION_BLOCK "I/O_FLT1"	// OB 82
TITLE = "I/O Point Fault"
VERSION : 0.1
VAR_TEMP
  OB82_EV_CLASS : BYTE ;	//16#39, Event class 3, Entering event state, Internal fault event
  OB82_FLT_ID : BYTE ;	//16#XX, Fault identifcation code
  OB82_PRIORITY : BYTE ;	//Priority of OB Execution
  OB82_OB_NUMBR : BYTE ;	//82 (Organization block 82, OB82)
  OB82_RESERVED_1 : BYTE ;	//Reserved for system
  OB82_IO_FLAG : BYTE ;	//Input (01010100), Output (01010101)
  OB82_MDL_ADDR : WORD ;	//Base address of module with fault
  OB82_MDL_DEFECT : BOOL ;	//Module defective
  OB82_INT_FAULT : BOOL ;	//Internal fault
  OB82_EXT_FAULT : BOOL ;	//External fault
  OB82_PNT_INFO : BOOL ;	//Point information
  OB82_EXT_VOLTAGE : BOOL ;	//External voltage low
  OB82_FLD_CONNCTR : BOOL ;	//Field wiring connector missing
  OB82_NO_CONFIG : BOOL ;	//Module has no configuration data
  OB82_CONFIG_ERR : BOOL ;	//Module has configuration error
  OB82_MDL_TYPE : BYTE ;	//Type of module
  OB82_SUB_MDL_ERR : BOOL ;	//Sub-Module is missing or has error
  OB82_COMM_FAULT : BOOL ;	//Communication fault
  OB82_MDL_STOP : BOOL ;	//Module is stopped
  OB82_WTCH_DOG_FLT : BOOL ;	//Watch dog timer stopped module
  OB82_INT_PS_FLT : BOOL ;	//Internal power supply fault
  OB82_PRIM_BATT_FLT : BOOL ;	//Primary battery is in fault
  OB82_BCKUP_BATT_FLT : BOOL ;	//Backup battery is in fault
  OB82_RESERVED_2 : BOOL ;	//Reserved for system
  OB82_RACK_FLT : BOOL ;	//Rack fault, only for bus interface module
  OB82_PROC_FLT : BOOL ;	//Processor fault
  OB82_EPROM_FLT : BOOL ;	//EPROM fault
  OB82_RAM_FLT : BOOL ;	//RAM fault
  OB82_ADU_FLT : BOOL ;	//ADU fault
  OB82_FUSE_FLT : BOOL ;	//Fuse fault
  OB82_HW_INTR_FLT : BOOL ;	//Hardware interupt input in fault
  OB82_RESERVED_3 : BOOL ;	//Reserved for system
  OB82_DATE_TIME : DATE_AND_TIME ;	//Date and time OB82 started
END_VAR
BEGIN
// (block stored without names or comments; labels and parameter names are numbered)
END_ORGANIZATION_BLOCK

ORGANIZATION_BLOCK "I/O_FLT2"	// OB 83
TITLE = "I/O Point Fault"
VERSION : 0.1
VAR_TEMP
  OB83_EV_CLASS : BYTE ;	//16#38/39, Event class 3, module inserted/removed (8/9)
  OB83_FLT_ID : BYTE ;	//16#XX, Fault identifcation code
  OB83_PRIORITY : BYTE ;	//Priority of OB Execution
  OB83_OB_NUMBR : BYTE ;	//83 (Organization block 83, OB83)
  OB83_RESERVED_1 : BYTE ;	//Reserved for system
  OB83_MDL_ID : BYTE ;	//Input module (01010100), Output module (01010101)
  OB83_MDL_ADDR : WORD ;	//Base address of module with point fault
  OB83_RACK_NUM : INT ;	//Number of rack that has module with point fault
  OB83_MDL_TYPE : WORD ;	//Module type with point fault
  OB83_DATE_TIME : DATE_AND_TIME ;	//Date and time OB83 started
END_VAR
BEGIN
// (block stored without names or comments; labels and parameter names are numbered)
END_ORGANIZATION_BLOCK

ORGANIZATION_BLOCK "CPU_FLT"	// OB 84
TITLE = "CPU Fault"
VERSION : 0.1
VAR_TEMP
  OB84_EV_CLASS : BYTE ;	//16#38/39, Event class 3, module inserted/removed (8/9)
  OB84_FLT_ID : BYTE ;	//16#81, Fault identifcation code
  OB84_PRIORITY : BYTE ;	//Priority of OB Execution
  OB84_OB_NUMBR : BYTE ;	//84 (Organization block 84, OB84)
  OB84_RESERVED_1 : BYTE ;	//Reserved for system
  OB84_RESERVED_2 : BYTE ;	//Reserved for system
  OB84_RESERVED_3 : WORD ;	//Reserved for system
  OB84_RESERVED_4 : DWORD ;	//Reserved for system
  OB84_DATE_TIME : DATE_AND_TIME ;	//Date and time OB84 started
END_VAR
BEGIN
// (block stored without names or comments; labels and parameter names are numbered)
END_ORGANIZATION_BLOCK

ORGANIZATION_BLOCK "OBNL_FLT"	// OB 85
TITLE = "Organization Block (OB) Not Loaded Fault"
VERSION : 0.1
VAR_TEMP
  OB85_EV_CLASS : BYTE ;	//16#35 Event class 3
  OB85_FLT_ID : BYTE ;	//16#XX, Fault identification code
  OB85_PRIORITY : BYTE ;	//Priority of OB Execution
  OB85_OB_NUMBR : BYTE ;	//85 (Organization block 85, OB85)
  OB85_RESERVED_1 : BYTE ;	//Reserved for system
  OB85_RESERVED_2 : BYTE ;	//Reserved for system
  OB85_RESERVED_3 : INT ;	//Reserved for system
  OB85_ERR_EV_CLASS : BYTE ;	//Class of event causing error
  OB85_ERR_EV_NUM : BYTE ;	//Number of event causing error
  OB85_OB_PRIOR : BYTE ;	//Priority of OB causing error
  OB85_OB_NUM : BYTE ;	//Number of OB causing error
  OB85_DATE_TIME : DATE_AND_TIME ;	//Date and time OB85 started
END_VAR
BEGIN
// (block stored without names or comments; labels and parameter names are numbered)
END_ORGANIZATION_BLOCK

ORGANIZATION_BLOCK "RACK_FLT"	// OB 86
TITLE = "Loss Of Rack Fault"
VERSION : 0.1
VAR_TEMP
  OB86_EV_CLASS : BYTE ;	//16#38/39 Event class 3
  OB86_FLT_ID : BYTE ;	//16#C1/C4/C5, Fault identifcation code
  OB86_PRIORITY : BYTE ;	//Priority of OB Execution
  OB86_OB_NUMBR : BYTE ;	//86 (Organization block 86, OB86)
  OB86_RESERVED_1 : BYTE ;	//Reserved for system
  OB86_RESERVED_2 : BYTE ;	//Reserved for system
  OB86_MDL_ADDR : WORD ;	//Base address of IM module in rack with fault
  OB86_RACKS_FLTD : ARRAY  [0 .. 31 ] OF BOOL ;	//Racks in fault
  OB86_DATE_TIME : DATE_AND_TIME ;	//Date and time OB86 started
END_VAR
BEGIN
// (block stored without names or comments; labels and parameter names are numbered)
END_ORGANIZATION_BLOCK

ORGANIZATION_BLOCK "COMM_FLT"	// OB 87
TITLE = "Communication Fault"
VERSION : 0.1
VAR_TEMP
  OB87_EV_CLASS : BYTE ;	//16#39 Event class 3
  OB87_FLT_ID : BYTE ;	//16#XX, Fault identifcation code
  OB87_PRIORITY : BYTE ;	//Priority of OB Execution
  OB87_OB_NUMBR : BYTE ;	//87 (Organization block 87, OB87)
  OB87_RESERVED_1 : BYTE ;	//Reserved for system
  OB87_RESERVED_2 : BYTE ;	//Reserved for system
  OB87_RESERVED_3 : WORD ;	//Reserved for system
  OB87_RESERVED_4 : DWORD ;	//Reserved for system
  OB87_DATE_TIME : DATE_AND_TIME ;	//Date and time OB87 started
END_VAR
BEGIN
// (block stored without names or comments; labels and parameter names are numbered)
END_ORGANIZATION_BLOCK

ORGANIZATION_BLOCK "COMPLETE RESTART"	// OB 100
TITLE = "Complete Restart"
VERSION : 0.1
VAR_TEMP
  OB100_EV_CLASS : BYTE ;	//16#13, Event class 1, Entering event state, Event logged in diagnostic buffer
  OB100_STRTUP : BYTE ;	//16#81/82/83/84 Method of startup
  OB100_PRIORITY : BYTE ;	//Priority of OB Execution
  OB100_OB_NUMBR : BYTE ;	//100 (Organization block 100, OB100)
  OB100_RESERVED_1 : BYTE ;	//Reserved for system
  OB100_RESERVED_2 : BYTE ;	//Reserved for system
  OB100_STOP : WORD ;	//Event that caused CPU to stop (16#4xxx)
  OB100_STRT_INFO : DWORD ;	//Information on how system started
  OB100_DATE_TIME : DATE_AND_TIME ;	//Date and time OB100 started
END_VAR
BEGIN
NETWORK
TITLE = Initialisiation of "MB_PNHCL"
//adapt the initialisation parameters according to your configuration
      L     1;
      T     DB1.DBW 0;
      L     2;
      T     DB1.DBW 2;
      L     T#5S;
      T     DB1.DBD 4;
      SET;
      S     DB1.DBX 8.0;
      CALL  FB 915 , DB 915 (
           DIW 0                    := DB1.DBW 0,
           DIW 2                    := DB1.DBW 2,
           DIW 8                    := 2,
           DID 10                   := DB1.DBD 4,
           DIX 14.0                 := DB1.DBX 8.0,
           DID 20                   := L#5000,
           DIW 26                   := 3,
           DIX 36.3                 := DB1.DBX 26.3,
           DIX 36.4                 := DB1.DBX 26.4,
           DIW 38                   := DB1.DBW 28,
           DIX 40.0                 := DB1.DBX 30.0,
           DIW 42                   := DB1.DBW 32,
           DIX 72.0                 := DB1.DBX 34.0,
           DIX 72.1                 := DB1.DBX 34.1,
           DIX 72.2                 := DB1.DBX 34.2);
      A     DB1.DBX 26.3;
      JCN   end;
      L     DB1.DBD 46;
      +     1;
      T     DB1.DBD 46;
      L     DB1.DBW 28;
      T     DB1.DBW 38;
      L     DB1.DBW 32;
      T     DB1.DBW 40;
end:  NOP   0;
END_ORGANIZATION_BLOCK

ORGANIZATION_BLOCK "PROG_ERR"	// OB 121
TITLE = "Programming Error"
VERSION : 0.1
VAR_TEMP
  OB121_EV_CLASS : BYTE ;	//16#25, Event class 2, Entering event state, Internal fault event
  OB121_SW_FLT : BYTE ;	//16#XX Software programming fault
  OB121_PRIORITY : BYTE ;	//Priority of OB Execution
  OB121_OB_NUMBR : BYTE ;	//121 (Organization block 121, OB121)
  OB121_BLK_TYPE : BYTE ;	//16#88/8A/8B/8C/8E Type of block fault occured in
  OB121_RESERVED_1 : BYTE ;	//Reserved for system
  OB121_FLT_REG : WORD ;	//16#XX Specific register that caused fault
  OB121_BLK_NUM : WORD ;	//Number of block that programming fault occured in
  OB121_PRG_ADDR : WORD ;	//Address in block where programming fault occured
  OB121_DATE_TIME : DATE_AND_TIME ;	//Date and time OB121 started
END_VAR
BEGIN
NETWORK
TITLE =
END_ORGANIZATION_BLOCK

ORGANIZATION_BLOCK "MOD_ERR"	// OB 122
TITLE = "Module Access Error"
VERSION : 0.1
VAR_TEMP
  OB122_EV_CLASS : BYTE ;	//16#29, Event class 2, Entering event state, Internal fault event
  OB122_SW_FLT : BYTE ;	//16#XX Software error code
  OB122_PRIORITY : BYTE ;	//Priority of OB Execution
  OB122_OB_NUMBR : BYTE ;	//122 (Organization block 122, OB122)
  OB122_BLK_TYPE : BYTE ;	//16#88/8C/8E Type of block fault occured in
  OB122_MEM_AREA : BYTE ;	//Memory area where access error occured
  OB122_MEM_ADDR : WORD ;	//Memory address where access error occured
  OB122_BLK_NUM : WORD ;	//Block number in which error occured
  OB122_PRG_ADDR : WORD ;	//Program address where error occured
  OB122_DATE_TIME : DATE_AND_TIME ;	//Date and time OB1 started
END_VAR
BEGIN
// (block stored without names or comments; labels and parameter names are numbered)
END_ORGANIZATION_BLOCK

